	IF	Temp_Mirror.stat.lrTempK > cfg.lrTemp_Precooled	AND  
		Pressure_Cryo.stat.lrPressure >= cfg.lrPress_Atm  		THEN
		ctrl.bEnable_RepressCtrl	:= FALSE;
		// Disable Evacuation Valve control
		ctrl.bEnable_Evac	:= FALSE;
		M_SysLog('Re-pressurization complete. State is Warm-Pressurized.');
		stat.nState	:= E_CRYO_CTRL_STATE.WARM_PRESS;
	ELSIF NOT ctrl.bEnable_RepressCtrl THEN
		// Re-pressurization has been interrupted.
		// Go back to WARM_VACUUM state.
		M_SysLog('Re-pressurization interrupted. State is Warm-Vacuum.');
		stat.nState := E_CRYO_CTRL_STATE.WARM_VACUUM;
	END_IF
	M_SetStatus(stat.nState);	
	RETURN;
	
	
	/////////////////////////////////
	E_CRYO_CTRL_STATE.ERROR:
	/////////////////////////////////
	//
	// RESET the controller in order to try to clear error
	IF ctrl.bReset THEN
		ctrl.bReset	:= FALSE;	// Clear RESET flag
		// Goto NONE state
		stat.nState	:= E_CRYO_CTRL_STATE.NONE;
		M_SetStatus(stat.nState);	
	ELSIF NOT stat.bError  THEN
		// Goto NONE state
		stat.nState	:= E_CRYO_CTRL_STATE.NONE;
		M_SetStatus(stat.nState);	
	END_IF
	RETURN;

END_CASE
END_METHOD

METHOD M_SysLog
VAR_INPUT
	str:	STRING(80);
END_VAR
VAR
	i:	INT;
END_VAR
nLogPos	:= nLogPos + 1;
IF nLogPos > 9 THEN
	FOR i := 1 TO 9 DO
		// Shift last 9 readings
		ptrLog[i-1]^ := ptrLog[i]^;
	END_FOR
	nLogPos	:= 9;
END_IF

ptrLog[nLogPos]^ := str;
END_METHOD

END_FUNCTION_BLOCK

// ---- POUs/Actuators/FB_CRYO_LN2_CTRL.TcPOU
FUNCTION_BLOCK FB_CRYO_LN2_CTRL EXTENDS FB_CRYO_BIN_CTRL
VAR_INPUT
	in_lrTempK:		LREAL;			// Temperature input value [K]
	in_bValid:		BOOL := TRUE;	// Temperature Valid flag
	// Two parameters for decision making
	in_lrTempValveOpen:		LREAL := 91.27;		// Open  valve if temperature above this value [K]
	in_lrTempValveClose:	LREAL := 79.148;	// Close valve if temperature below this value [K]
END_VAR
VAR_OUTPUT
END_VAR
VAR
END_VAR

// Check the validity of the temperature reading.
// Start the check after 200 cycles.
IF stat.nCycleCounter > 200 THEN
	IF NOT in_bValid THEN
		// The temperature is not valid. 
		// The controller cannot work.
		stat.bCtrlOK	:= FALSE;
	ELSIF in_lrTempValveClose >= in_lrTempValveOpen THEN
		// Wrong configuration.
		// ValveClose MUST be lower than ValveOpen temperature
		stat.bCtrlOK	:= FALSE;
	ELSE
		// The temperature is valid. 
		stat.bCtrlOK	:= TRUE;
	END_IF
ELSE
	// The temperature is valid. 
	stat.bCtrlOK	:= TRUE;
END_IF

// Execute parent FB.
SUPER^();

METHOD M_SetStatus
VAR_INPUT
	nState:	E_CRYO_BIN_CTRL_STATE;
END_VAR
// Execute the status of the parent FB
SUPER^.M_SetStatus(nState);

// Set proper error description, if any.
IF Actuator.stat.bError THEN
	stat.sState	:= 'Valve failure';
ELSIF NOT stat.bCtrlOK THEN
	stat.sState	:= 'Temperature not valid';
END_IF
END_METHOD

METHOD M_User_SetAction : INT
VAR_INPUT
END_VAR
// TODO USER
// Overwrite Method FB_CRYO_BIN_CTRL::M_User_SetOutput()
//
// This method implements the logic for controlling the LN2 valve.
// 
// FB_CRYO_LN2_CTRL input parameters:
//
// in_lrTempK          - LN2 temperature
// in_bValid           - Flag if temperature reading is valid
// in_lrTempValveOpen  - Temperature upper limit [K]. Valve opens  when:  LN2 > in_lrTempValveOpen
// in_lrTempValveClose - Temperature lower limit [K]. Valve closes when:  LN2 < in_lrTempValveClose
//
// in_lrTempValveOpen > in_lrTempValveClose, e.g. 91.27K > 79.148K.
//
	
IF	stat.nState = E_CRYO_BIN_CTRL_STATE.ACTIVE_OFF  OR  
	stat.nState = E_CRYO_BIN_CTRL_STATE.ACTIVE_ON THEN
	// Check if input temperature value is valid.
	// If OK, check temperature against the limits	
	IF NOT stat.bCtrlOK THEN
		// Temperature reading is not valid.
		// Dectivate the actuator, i.e. close the valve
		M_User_SetAction	:= E_CRYO_BIN_CTRL_ACTION.OFF;
		stat.nState	:= E_CRYO_BIN_CTRL_STATE.ERROR;
	ELSIF in_lrTempK > in_lrTempValveOpen THEN
		// Activate the actuator, i.e. open the valve
		M_User_SetAction	:= E_CRYO_BIN_CTRL_ACTION.ON;
	ELSIF in_lrTempK < in_lrTempValveClose THEN
		// Dectivate the actuator, i.e. close the valve
		M_User_SetAction	:= E_CRYO_BIN_CTRL_ACTION.OFF;
	END_IF
	
ELSE
	// Don't do anything
	M_User_SetAction	:= E_CRYO_BIN_CTRL_ACTION.NONE;
END_IF
END_METHOD

END_FUNCTION_BLOCK

// ---- POUs/Actuators/FB_CRYO_BIN_CTRL.TcPOU
// Binary Controller
FUNCTION_BLOCK FB_CRYO_BIN_CTRL
VAR_INPUT
	in_nFeedback:		E_CRYO_BIN_ACT_FEEDBACK := E_CRYO_BIN_ACT_FEEDBACK.ON_ONLY;	// Feedbacks
	in_nTimeout:		UDINT := 10000;	// Timeout for switching on/off [ms]. Default 10000.
	in_bActiveLowCtrl:	BOOL := FALSE;	// Active Low for Control output
	in_bActiveLowStat:	BOOL := FALSE;	// Active Low for Status signals, i.e. feedback
	in_bEnable:			BOOL := FALSE;	// Controller active while in_bEnable is TRUE
END_VAR
VAR
	
	{attribute 'OPC.UA.DA' := '1'}
	Actuator:	FB_CRYO_BIN_ACT;	// Heater, valve, etc.
	
	stat:		T_CRYO_BIN_CTRL_STATUS;


	{attribute 'OPC.UA.DA' := '0'}
	bReset:		BOOL := FALSE;		// RESET Command


	{attribute 'OPC.UA.DA' := '0'}
	timer:		TON;		// Timer for commands
	
	
END_VAR

// Increment cycle counter
stat.nCycleCounter := stat.nCycleCounter + 1;

// Execute Actuator FB on every cycle
Actuator(
	in_nFeedback		:= in_nFeedback,
	in_nTimeout			:= in_nTimeout,
	in_bActiveLowCtrl	:= in_bActiveLowCtrl,
	in_bActiveLowStat	:= in_bActiveLowStat);


CASE stat.nState OF
	/////////////////////////////////
	E_CRYO_BIN_CTRL_STATE.NONE:
	/////////////////////////////////
	//
	// This is the state on power-up.
	// Determine the initial state based on the command amd actuator state.
	IF Actuator.stat.bError  OR NOT stat.bCtrlOK	THEN
		stat.nState	:= E_CRYO_BIN_CTRL_STATE.ERROR;
	ELSIF in_bEnable  AND  Actuator.stat.bON	THEN
		stat.nState	:= E_CRYO_BIN_CTRL_STATE.ACTIVE_ON;
	ELSIF in_bEnable  AND  Actuator.stat.bOFF	THEN
		stat.nState	:= E_CRYO_BIN_CTRL_STATE.ACTIVE_OFF;
	ELSIF NOT in_bEnable  THEN
		stat.nState	:= E_CRYO_BIN_CTRL_STATE.OFF;
	END_IF
	M_SetStatus(stat.nState);	
	RETURN;
	

	/////////////////////////////////
	E_CRYO_BIN_CTRL_STATE.OFF:
	/////////////////////////////////
	//
	IF	Actuator.stat.bError	OR NOT stat.bCtrlOK	THEN
		stat.nState	:= E_CRYO_BIN_CTRL_STATE.ERROR;
	ELSIF in_bEnable  THEN
		// Activate the control loop.
		// Goto Active_Off first.
		//
		// Start the timer
		timer(IN:=FALSE);
		timer(IN:=TRUE, PT:=UDINT_TO_TIME(in_nTimeout));
		// Set next state
		stat.nState	:= E_CRYO_BIN_CTRL_STATE.ACTIVE_OFF;
	END_IF
	M_SetStatus(stat.nState);	
	RETURN;
	
	
	/////////////////////////////////
	E_CRYO_BIN_CTRL_STATE.ACTIVE_OFF:
	/////////////////////////////////
	//
	IF	Actuator.stat.bError	OR NOT stat.bCtrlOK  THEN
		stat.nState	:= E_CRYO_BIN_CTRL_STATE.ERROR;
	ELSIF NOT in_bEnable  THEN
		// Goto Off.
		//
		// Set next state
		stat.nState	:= E_CRYO_BIN_CTRL_STATE.OFF;
	ELSIF M_User_SetAction() = E_CRYO_BIN_CTRL_ACTION.ON THEN
		// Goto Active_Off.
		//
		// Start the timer
		timer(IN:=FALSE);
		timer(IN:=TRUE, PT:=UDINT_TO_TIME(in_nTimeout));
		
		// Trigger action
		Actuator(in_bExecute:=FALSE);
		Actuator(in_bExecute:=TRUE, in_nCommand:=E_CRYO_BIN_ACT_CMD.ON);
		
		// Set next state
		stat.nState	:= E_CRYO_BIN_CTRL_STATE.ACTIVE_SWITCHING_ON;
	END_IF
	M_SetStatus(stat.nState);	
	RETURN;
	
	
	//////////////////////////////////////////
	E_CRYO_BIN_CTRL_STATE.ACTIVE_SWITCHING_ON:
	//////////////////////////////////////////
	//
	// Check for timeout
	timer(IN:=TRUE);
	IF timer.Q THEN
		// Stop the timer
		timer(IN:=FALSE);
		// Goto ERROR state
		stat.nState	:= E_CRYO_BIN_CTRL_STATE.ERROR;
	ELSIF	Actuator.stat.bError	THEN
		stat.nState	:= E_CRYO_BIN_CTRL_STATE.ERROR;
	ELSIF Actuator.stat.bON THEN
		// The actuator is ON, transition completed.
		// Goto Active_On.
		stat.nState	:= E_CRYO_BIN_CTRL_STATE.ACTIVE_ON;
	END_IF
	M_SetStatus(stat.nState);	
	RETURN;
	

	/////////////////////////////////
	E_CRYO_BIN_CTRL_STATE.ACTIVE_ON:
	/////////////////////////////////
	//
	IF	Actuator.stat.bError	THEN
		stat.nState	:= E_CRYO_BIN_CTRL_STATE.ERROR;
	ELSIF	NOT in_bEnable 		OR  
			NOT stat.bCtrlOK	OR
			M_User_SetAction() = E_CRYO_BIN_CTRL_ACTION.OFF THEN
		// Goto Active_Off.
		// If NOT in_bExecute, the system will continue to complete OFF
		//
		// Start the timer
		timer(IN:=FALSE);
		timer(IN:=TRUE, PT:=UDINT_TO_TIME(in_nTimeout));
		
		// Trigger action
		Actuator(in_bExecute:=FALSE);
		Actuator(in_bExecute:=TRUE, in_nCommand:=E_CRYO_BIN_ACT_CMD.OFF);
		
		// Set next state
		stat.nState	:= E_CRYO_BIN_CTRL_STATE.ACTIVE_SWITCHING_OFF;
	END_IF
	M_SetStatus(stat.nState);	
	RETURN;
	
	
	///////////////////////////////////////////
	E_CRYO_BIN_CTRL_STATE.ACTIVE_SWITCHING_OFF:
	///////////////////////////////////////////
	//
	// Check for timeout
	timer(IN:=TRUE);
	IF timer.Q THEN
		// Stop the timer
		timer(IN:=FALSE);
		// Goto ERROR state
		stat.nState	:= E_CRYO_BIN_CTRL_STATE.ERROR;
	ELSIF	Actuator.stat.bError	THEN
		stat.nState	:= E_CRYO_BIN_CTRL_STATE.ERROR;
	ELSIF Actuator.stat.bOFF THEN
		// The actuator is OFF, transition completed.
		// Goto Active_Off.
		stat.nState	:= E_CRYO_BIN_CTRL_STATE.ACTIVE_OFF;
	END_IF
	M_SetStatus(stat.nState);	
	RETURN;
	
	/////////////////////////////////
	E_CRYO_BIN_CTRL_STATE.ERROR:
	/////////////////////////////////
	//
	M_User_TryRecovery();

END_CASE

METHOD M_Reset
VAR_INPUT
END_VAR
// By setting the bReset flag,
// The actuator will try to exit error state.
// In ERROR state, method M_User_TryRecovery() is executed.
bReset	:= TRUE;
END_METHOD

METHOD M_SetStatus
VAR_INPUT
	nState:	E_CRYO_BIN_CTRL_STATE;
END_VAR
stat.bActON		:= Actuator.stat.bON;
stat.bActOFF	:= Actuator.stat.bOFF;


CASE nState OF
	
	E_CRYO_BIN_CTRL_STATE.OFF:
	stat.bDone	:= TRUE;
	stat.bBusy	:= FALSE;
	stat.bError	:= FALSE;
	stat.bActive:= FALSE;
	stat.sState	:= 'OFF';
	
	E_CRYO_BIN_CTRL_STATE.ACTIVE_OFF:
	stat.bDone	:= TRUE;
	stat.bBusy	:= FALSE;
	stat.bError	:= FALSE;
	stat.bActive:= TRUE;
	stat.sState	:= 'ACTIVE_OFF';
	
	E_CRYO_BIN_CTRL_STATE.ACTIVE_ON:
	stat.bDone	:= TRUE;
	stat.bBusy	:= FALSE;
	stat.bError	:= FALSE;
	stat.bActive:= TRUE;
	stat.sState	:= 'ACTIVE_ON';
	
	E_CRYO_BIN_CTRL_STATE.ACTIVE_SWITCHING_ON:
	stat.bDone	:= FALSE;
	stat.bBusy	:= TRUE;
	stat.bError	:= FALSE;
	stat.bActive:= TRUE;
	stat.sState	:= 'ACTIVE_SWITCHING_ON...';
	
	E_CRYO_BIN_CTRL_STATE.ACTIVE_SWITCHING_OFF:
	stat.bDone	:= FALSE;
	stat.bBusy	:= TRUE;
	stat.bError	:= FALSE;
	stat.bActive:= TRUE;
	stat.sState	:= 'ACTIVE_SWITCHING_OFF...';
	
	E_CRYO_BIN_CTRL_STATE.ERROR:
	stat.bDone	:= TRUE;
	stat.bBusy	:= FALSE;
	stat.bError	:= TRUE;
	stat.bActive:= FALSE;
	stat.sState	:= 'ERROR';

END_CASE
END_METHOD

METHOD M_User_SetAction : INT
VAR_INPUT
END_VAR
// TODO USER
//
// This method implements the logic for controlling the actuator.
// The actuator can be a heater, valve, etc.
// There are two input values from sensors and two deltas for comparison.
//
// This example implements the heater control with the following assumptions:
//
// in_lrInput1 - Temperature of the Cryo Bench (B)
// in_lrInput2 - Temperature of the Detector (D). Coming from Lakeshore.
// in_lrPar1 - Delta [K] to turn the heater ON:  IF B < D - in_lrPar1
// in_lrPar2 - Delta [K] to turn the heater OFF: IF B > D - in_lrPar2
//
// in_lrDelta1 > in_lrDelta2, e.g. 10K > 4K.
//
IF	stat.nState = E_CRYO_BIN_CTRL_STATE.ACTIVE_OFF  OR  
	stat.nState = E_CRYO_BIN_CTRL_STATE.ACTIVE_ON THEN
(*	
	IF in_lrInput1 < in_lrInput2 - in_lrPar1 THEN
		// Activate the actuator
		M_User_SetOutput	:= E_CRYO_BIN_CTRL_ACTION.ON;
	ELSIF in_lrInput1 > in_lrInput2 - in_lrPar2 THEN
		// Dectivate the actuator
		M_User_SetOutput	:= E_CRYO_BIN_CTRL_ACTION.OFF;
	END_IF
*)
ELSE
	// Don't do anything
	M_User_SetAction	:= E_CRYO_BIN_CTRL_ACTION.NONE;
END_IF
END_METHOD

METHOD M_User_TryRecovery
VAR_INPUT
END_VAR
// TODO USER
// This is the default recovery routine.
// To be customided by the user, if needed.
//
IF bReset THEN
	// RESET the controller in order to try to clear error
	bReset	:= FALSE;	// Clear RESET flag
	
	// Start the timer
	timer(IN:=FALSE);
	timer(IN:=TRUE, PT:=T#5S);
	
	// Trigger action
	Actuator(in_bExecute:=FALSE);
	Actuator(in_bExecute:=TRUE, in_nCommand:=E_CRYO_BIN_ACT_CMD.OFF);
	
	// Goto SWITCHING_OFF state
	stat.nState	:= E_CRYO_BIN_CTRL_STATE.ACTIVE_SWITCHING_OFF;
	M_SetStatus(stat.nState);	
ELSIF NOT Actuator.stat.bError AND stat.bCtrlOK  THEN
	// Self recovery since everything seems to be OK now.
	// Goto NONE state.
	// From there proper state will be found and set.
	stat.nState	:= E_CRYO_BIN_CTRL_STATE.NONE;
	M_SetStatus(stat.nState);	
END_IF
END_METHOD

END_FUNCTION_BLOCK

// ---- POUs/Actuators/FB_CRYO_BIN_ACT.TcPOU
FUNCTION_BLOCK FB_CRYO_BIN_ACT
VAR_INPUT
	in_nFeedback:		E_CRYO_BIN_ACT_FEEDBACK := E_CRYO_BIN_ACT_FEEDBACK.ON_ONLY;	// Feedback configuration.
	in_nTimeout:		UDINT := 10000;	// Timeout for switching on/off [ms]. Default 10000.
	in_bActiveLowCtrl:	BOOL := FALSE;	// Active Low for Control output
	in_bActiveLowStat:	BOOL := FALSE;	// Active Low for Status signals, i.e. feedback
	in_nCommand:		E_CRYO_BIN_ACT_CMD	:= E_CRYO_BIN_ACT_CMD.NONE;	// Command
	in_bExecute:		BOOL := FALSE;	// Execute trigger
END_VAR
VAR
	{attribute 'OPC.UA.DA' := '0'}
	i_nCouplerState	AT%I*:	UINT;		// Terminal state. Should be 8, i.e. OP.
	{attribute 'OPC.UA.DA' := '0'}
	i_bON			AT%I*:	BOOL;		// Feedback for ON
	{attribute 'OPC.UA.DA' := '0'}
	i_bOFF			AT%I*:	BOOL;		// Feedback for OFF
	
	{attribute 'OPC.UA.DA' := '0'}
	q_bCtrl			AT%Q*:	BOOL;		// Control output signal
	
	stat:		T_CRYO_BIN_ACT_STATUS;

	
	{attribute 'OPC.UA.DA' := '0'}
	timer:		TON;		// Timer for commands
	{attribute 'OPC.UA.DA' := '0'}
	trigCMD:	R_TRIG;		// Trigger for new command
	
	{attribute 'OPC.UA.DA' := '0'}
	nCommand:	E_CRYO_BIN_ACT_CMD	:= E_CRYO_BIN_ACT_CMD.NONE;	// Command

END_VAR

// Get the feedback
M_GetFeedback();

// Check for new command
trigCMD(CLK:=in_bExecute);
IF trigCMD.Q THEN
	nCommand			:= in_nCommand;
	stat.nLastCommand	:= in_nCommand;
ELSE
	nCommand		:= E_CRYO_BIN_ACT_CMD.NONE;
END_IF

// If the system is not operational, this is an error.
IF i_nCouplerState <> 8 THEN
	stat.nState	:= E_CRYO_BIN_ACT_STATE.ERROR;
	stat.sState	:= 'ERROR: System not OPERATIONAL';
	M_SetStatus(stat.nState);	
END_IF

CASE stat.nState OF
	/////////////////////////////////
	E_CRYO_BIN_ACT_STATE.NONE:
	/////////////////////////////////
	//
	// Determine the initial state based on the feedback
	IF stat.bON	THEN
		stat.nState	:= E_CRYO_BIN_ACT_STATE.ON;
	ELSIF stat.bOFF	THEN
		stat.nState	:= E_CRYO_BIN_ACT_STATE.OFF;
	ELSE
		stat.nState	:= E_CRYO_BIN_ACT_STATE.ERROR;
		stat.sState	:= 'ERROR';
	END_IF
	M_SetStatus(stat.nState);	
	RETURN;
	

	/////////////////////////////////
	E_CRYO_BIN_ACT_STATE.OFF:
	/////////////////////////////////
	//
	IF	stat.bON  OR  
		stat.bError	THEN
		// This should never happen in state OFF
		stat.nState	:= E_CRYO_BIN_ACT_STATE.ERROR;
		stat.sState	:= 'ERROR: Lost ON state.';
		M_SetStatus(stat.nState);	
	ELSE
		// Check for command to go ON
		IF nCommand = E_CRYO_BIN_ACT_CMD.ON THEN
			// Start the timer
			timer(IN:=FALSE);
			timer(IN:=TRUE, PT:=UDINT_TO_TIME(in_nTimeout));
			// Activate the output
			M_SetCtrlOutput(TRUE);
			// Goto SWITCHING_ON state
			stat.nState	:= E_CRYO_BIN_ACT_STATE.SWITCHING_ON;
			M_SetStatus(stat.nState);	
		END_IF
	END_IF
	RETURN;
	
	
	/////////////////////////////////
	E_CRYO_BIN_ACT_STATE.SWITCHING_ON:
	/////////////////////////////////
	//
	// Check for timeout
	timer(IN:=TRUE);
	IF timer.Q THEN
		// Stop the timer
		timer(IN:=FALSE);
		// Goto ERROR state
		stat.nState	:= E_CRYO_BIN_ACT_STATE.ERROR;
		stat.sState	:= 'ERROR: Timeout switching ON';
		M_SetStatus(stat.nState);	
		RETURN;
	END_IF
	
	// Check if we have reached ON state
	IF stat.bON	AND NOT stat.bOFF	THEN
		// Stop the timer
		timer(IN:=FALSE);
		// Goto ON state
		stat.nState	:= E_CRYO_BIN_ACT_STATE.ON;
		M_SetStatus(stat.nState);	
	END_IF
	RETURN;
	

	/////////////////////////////////
	E_CRYO_BIN_ACT_STATE.ON:
	/////////////////////////////////
	//
	IF	stat.bOFF  OR  
		stat.bError	THEN
		// This should never happen in state ON
		stat.nState	:= E_CRYO_BIN_ACT_STATE.ERROR;
		stat.sState	:= 'ERROR: Lost OFF state.';
		M_SetStatus(stat.nState);	
	ELSE
		// Check for command to go OFF
		IF nCommand = E_CRYO_BIN_ACT_CMD.OFF THEN
			// Start the timer
			timer(IN:=FALSE);
			timer(IN:=TRUE, PT:=UDINT_TO_TIME(in_nTimeout));
			// Deactivate the output
			M_SetCtrlOutput(FALSE);
			// Goto SWITCHING_OFF state
			stat.nState	:= E_CRYO_BIN_ACT_STATE.SWITCHING_OFF;
			M_SetStatus(stat.nState);	
		END_IF
	END_IF
	RETURN;
	
	
	//////////////////////////////////
	E_CRYO_BIN_ACT_STATE.SWITCHING_OFF:
	//////////////////////////////////
	//
	// Check for timeout
	timer(IN:=TRUE);
	IF timer.Q THEN
		// Stop the timer
		timer(IN:=FALSE);
		// Goto ERROR state
		stat.nState	:= E_CRYO_BIN_ACT_STATE.ERROR;
		stat.sState	:= 'ERROR: Timeout switching OFF';
		M_SetStatus(stat.nState);	
		RETURN;
	END_IF
	
	// Check if we have reached OFF state
	IF stat.bOFF AND NOT stat.bON	THEN
		// Stop the timer
		timer(IN:=FALSE);
		// Goto OFF state
		stat.nState	:= E_CRYO_BIN_ACT_STATE.OFF;
		M_SetStatus(stat.nState);	
	END_IF
	RETURN;
	
	/////////////////////////////////
	E_CRYO_BIN_ACT_STATE.ERROR:
	/////////////////////////////////
	//
	// Deactivate the output
	M_SetCtrlOutput(FALSE);
	
	// Check for command to go ON
	IF nCommand = E_CRYO_BIN_ACT_CMD.ON THEN
		// Start the timer
		timer(IN:=FALSE);
		timer(IN:=TRUE, PT:=UDINT_TO_TIME(in_nTimeout));
		// Activate the output
		M_SetCtrlOutput(TRUE);
		// Goto SWITCHING_ON state
		stat.nState	:= E_CRYO_BIN_ACT_STATE.SWITCHING_ON;
		M_SetStatus(stat.nState);	
	// Check for command to go OFF
	ELSIF nCommand = E_CRYO_BIN_ACT_CMD.OFF THEN
		// Start the timer
		timer(IN:=FALSE);
		timer(IN:=TRUE, PT:=UDINT_TO_TIME(in_nTimeout));
		// Deactivate the output
		M_SetCtrlOutput(FALSE);
		// Goto SWITCHING_OFF state
		stat.nState	:= E_CRYO_BIN_ACT_STATE.SWITCHING_OFF;
		M_SetStatus(stat.nState);	
	END_IF
	RETURN;

END_CASE

METHOD M_GetFeedback
VAR_INPUT
END_VAR
// Get ON/OFF status based on active low configuration
IF in_bActiveLowStat	THEN
	stat.bON	:= NOT i_bON;
	stat.bOFF	:= NOT i_bOFF;
ELSE
	stat.bON	:= i_bON;
	stat.bOFF	:= i_bOFF;
END_IF

// Check for possible feedback errors.
// Also, adjust the OFF signal, if only ON feedback exists.
IF in_nFeedback = E_CRYO_BIN_ACT_FEEDBACK.ON_AND_OFF  THEN
	// There are separate signals for ON and OFF.
	// The status is already properly assigned. Nothing more to do.
	// If both feedback signals are active, this is an error.
	(*
	IF stat.bON AND stat.bOFF	THEN
		stat.nState	:= E_CRYO_BIN_ACT_STATE.ERROR;
		stat.sState	:= 'ERROR: Both ON and OFF signals active!';
		M_SetStatus(stat.nState);	
	END_IF
	*)
	;
ELSIF in_nFeedback = E_CRYO_BIN_ACT_FEEDBACK.ON_ONLY  THEN
	// There is only a feedback signal for ON.
	// Therefore, stat.bOFF := NOT stat.bON
	stat.bOFF	:= NOT stat.bON;
END_IF
END_METHOD

METHOD M_SetCtrlOutput
VAR_INPUT
	in_bSignal:	BOOL;
END_VAR
// Set control output signal based on active low configuration
IF in_bActiveLowCtrl	THEN
	q_bCtrl	:= NOT in_bSignal;
ELSE
	q_bCtrl	:= in_bSignal;
END_IF
END_METHOD

METHOD M_SetStatus
VAR_INPUT
	nState:	E_CRYO_BIN_ACT_STATE;
END_VAR
CASE stat.nState OF
	
	E_CRYO_BIN_ACT_STATE.OFF,
	E_CRYO_BIN_ACT_STATE.ON:
	stat.bDone	:= TRUE;
	stat.bBusy	:= FALSE;
	stat.bError	:= FALSE;
	
	E_CRYO_BIN_ACT_STATE.SWITCHING_ON,
	E_CRYO_BIN_ACT_STATE.SWITCHING_OFF:
	stat.bDone	:= FALSE;
	stat.bBusy	:= TRUE;
	stat.bError	:= FALSE;
	
	E_CRYO_BIN_ACT_STATE.ERROR:
	stat.bDone	:= TRUE;
	stat.bBusy	:= FALSE;
	stat.bError	:= TRUE;
END_CASE

// Set status string
CASE stat.nState OF
	
	E_CRYO_BIN_ACT_STATE.OFF:
	stat.sState	:= 'OFF';
	
	E_CRYO_BIN_ACT_STATE.ON:
	stat.sState	:= 'ON';
	
	E_CRYO_BIN_ACT_STATE.SWITCHING_ON:
	stat.sState	:= 'SWITCHING_ON...';
	
	E_CRYO_BIN_ACT_STATE.SWITCHING_OFF:
	stat.sState	:= 'SWITCHING_OFF...';
	
	E_CRYO_BIN_ACT_STATE.ERROR:
	// Error string was set where the error was detected.
	//	stat.sState	:= 'ERROR';
	;
END_CASE
END_METHOD

END_FUNCTION_BLOCK

// ---- POUs/Actuators/FB_CRYO_VALVE_CTRL.TcPOU
FUNCTION_BLOCK FB_CRYO_VALVE_CTRL EXTENDS FB_CRYO_BIN_CTRL
VAR_INPUT
END_VAR
VAR_OUTPUT
END_VAR
VAR
END_VAR

// Execute parent FB.
SUPER^();

METHOD M_SetStatus
VAR_INPUT
	nState:	E_CRYO_BIN_CTRL_STATE;
END_VAR
// Execute the status of the parent FB
SUPER^.M_SetStatus(nState);

// Set proper error description, if any.
IF Actuator.stat.bError THEN
	stat.sState	:= 'Valve failure';
END_IF
END_METHOD

METHOD M_User_SetAction : INT
VAR_INPUT
END_VAR
// TODO USER
// Set Valve command based on the input parameter in_bEnable.
//
	
IF	stat.nState = E_CRYO_BIN_CTRL_STATE.ACTIVE_OFF  AND in_bEnable THEN
	// Activate the actuator, i.e. open the valve
	M_User_SetAction	:= E_CRYO_BIN_CTRL_ACTION.ON;
ELSIF  stat.nState = E_CRYO_BIN_CTRL_STATE.ACTIVE_ON AND NOT in_bEnable THEN
	// Dectivate the actuator, i.e. close the valve
	M_User_SetAction	:= E_CRYO_BIN_CTRL_ACTION.OFF;
ELSE
	// Don't do anything
	M_User_SetAction	:= E_CRYO_BIN_CTRL_ACTION.NONE;
END_IF
END_METHOD

END_FUNCTION_BLOCK

// ---- POUs/Subsystems/Evacuation/FB_CRYO_EVACUATION_SYSTEM.TcPOU
//
// Evacuation System Controller.
// The system consists of:
// - Evacuation Valve
// - Root Pump
// - Turbo Pump
//
FUNCTION_BLOCK FB_CRYO_EVACUATION_SYSTEM
VAR_INPUT
	in_Cryo_Cfg:			T_CRYO_CFG;					// Cryo configuration
	in_Temp_Cryo:			T_CRYO_TEMPERATURE_STATUS;	// Cold Bench temperature	
	in_Pressure_Cryo:		T_CRYO_PRESSURE_STATUS;		// Cryostat Pressure
	in_Pressure_Evac:		T_CRYO_PRESSURE_STATUS;		// Evacuation Pressure
	
	in_bRepressValveOpen:	BOOL;	// Repressure Valve Open flag
	in_bRepressValveOK:		BOOL;	// Repressure Valve OK flag
	in_nFeedback:	E_CRYO_BIN_ACT_FEEDBACK := E_CRYO_BIN_ACT_FEEDBACK.ON_ONLY;	// Feedbacks
	// Time between closing Vac valve and Switching OFF the vac Pump [ms]
	in_nTimeout:	UDINT := 3200;	// Timeout for switching on/off [ms]
	in_bEnable:		BOOL := FALSE;	// Controller active while in_bEnable is TRUE
	in_bCmd:		BOOL := FALSE;	// ON=TRUE, OFF=FALSE
END_VAR
VAR
	
	{attribute 'OPC.UA.DA' := '0'}
	i_bRootPumpOn	AT%I*:	BOOL;		// Root Pump Feedback
	{attribute 'OPC.UA.DA' := '0'}
	i_bTurboPumpOn	AT%I*:	BOOL;		// Turbo Pump Feedback
	
	{attribute 'OPC.UA.DA' := '0'}
	q_bPumpCtrl		AT%Q*:	BOOL;			// Pump Control signal
	
	stat:			T_CRYO_EVACUATION_SYSTEM_STATUS;

	{attribute 'OPC.UA.DA' := '1'}
	Valve:	FB_CRYO_BIN_ACT;			// Evacuation Valve 

	{attribute 'OPC.UA.DA' := '0'}
	bExecute_Valve:	BOOL := FALSE;

	{attribute 'OPC.UA.DA' := '0'}
	nCommand_Valve:	E_CRYO_BIN_ACT_CMD	:= E_CRYO_BIN_ACT_CMD.NONE;	// Command

	{attribute 'OPC.UA.DA' := '0'}
	bReset:		BOOL := FALSE;		// RESET Command

	{attribute 'OPC.UA.DA' := '0'}
	bValveCmd:	BOOL := FALSE;		// Valve Command - TRUE=OPEN, FALSE=CLOSE


	{attribute 'OPC.UA.DA' := '0'}
	timerTurbo:	TON;		// Timer for Turbo Pump
	
	{attribute 'OPC.UA.DA' := '0'}
	timerValveDelay:	TON;		// Timer for measuring time after Valve is closed
	
	{attribute 'OPC.UA.DA' := '0'}
	timerValveCtrl:	TON;		// Timer for Valve open/close timeout
	
	{attribute 'OPC.UA.DA' := '0'}
	trigEnable:	R_TRIG;			// Trigger for in_bEnable
	
	{attribute 'OPC.UA.DA' := '0'}
	trigDisable:F_TRIG;			// Trigger for in_bEnable=FALSE, i.e. Disable
	
	{attribute 'OPC.UA.DA' := '0'}
	trigTurbo:	R_TRIG;		// Trigger for start of TurboPump
	
	{attribute 'OPC.UA.DA' := '0'}
	trigValveClosed:	R_TRIG;		// Trigger for Valve Closed. Start timerValve on trigger.
	
END_VAR

// Increment cycle counter
stat.nCycleCounter := stat.nCycleCounter + 1;

// Pump control based on Valve status.
M_PumpCtrl();

// Check for errors
M_CheckErrors();

// Get Valve Command based on pressure and temperature conditions
M_SetValveCommand();


// Execute Valve FB on every cycle
Valve(	in_bExecute	:= bExecute_Valve,
		in_nCommand	:= nCommand_Valve,
		in_nFeedback:= in_nFeedback);


M_StateMachine();

METHOD M_CheckErrors
VAR_INPUT
END_VAR
VAR
END_VAR
// TODO: Set stat.sStatus for each failure
IF Valve.stat.bON  AND  (in_bRepressValveOpen  OR  NOT in_bRepressValveOK) THEN
	// Emergency situation. Close the Valve
	stat.bEmergency	:= TRUE;
	stat.bError	:= TRUE;
ELSIF stat.bEnabled  AND  (in_bRepressValveOpen  OR  NOT in_bRepressValveOK) THEN
	// The Evacuation system should never be enabled 
	// if there is a problem with the repressurizing valve.
	// Emergency situation. Do not operate.
	stat.bEmergency	:= TRUE;
	stat.bError	:= TRUE;
ELSIF NOT in_bRepressValveOK THEN
	stat.bError	:= TRUE;
ELSIF NOT in_Pressure_Cryo.bValid THEN
	stat.bError	:= TRUE;
ELSIF NOT in_Pressure_Evac.bValid THEN
	stat.bError	:= TRUE;
ELSIF Valve.stat.bError THEN
	stat.bError	:= TRUE;
ELSE
	stat.bError	:= FALSE;
END_IF

// Additional check for emergency situation.
// If there is an error while the Evacuation Valve is open, close it immediately.
IF stat.bError  AND  Valve.stat.bON  THEN
	stat.bEmergency	:= TRUE;
END_IF

IF stat.bError  THEN
	stat.bEnabled	:= FALSE;	// Disable Evacuation System
END_IF
END_METHOD

// Pump control based on Valve status.
METHOD M_PumpCtrl
VAR_INPUT
END_VAR
//
// Capture in_bEnable going TRUE.
// When it happens, start the pumps by activating the control output.
//
trigEnable(CLK:=in_bEnable);
IF trigEnable.Q THEN
	stat.bEnabled	:= TRUE;
	stat.bEmergency	:= FALSE;	// Clear emergency warning, if any
	stat.bError		:= FALSE;	// Clear error
	q_bPumpCtrl		:= TRUE;	// Start pumps
ELSIF NOT in_bEnable THEN
	stat.bEnabled		:= FALSE;
END_IF


//
// Set the status of the Root Pump
//
stat.bRootPumpON	:= i_bRootPumpOn;


//
// Set the status of the Turbo Pump
//
IF i_bTurboPumpOn THEN
	// Turbo pump is running.
	stat.bTurboPumpON	:= TRUE;
ELSE
	timerTurbo(IN:=FALSE);
	stat.bTurboPumpON		:= FALSE;
	stat.bTurboPump10min	:= FALSE;
END_IF



//
// Capture the moment when Turbo Pump started.
// Turbo Pump is fully operational after 10 min of operation (in_nTime_TurboPump).
//
// Execute timer for Turbo Pump
timerTurbo();

trigTurbo(CLK:=stat.bTurboPumpON);
IF trigTurbo.Q  THEN
	//
	// Turbo Pump has just started.
	// Start the timer that will signal that the turbo pump is fully operational.
	//
	// Reset the timer.
	timerTurbo(IN:=FALSE);
	// Start the timer for Turbo Pump warmup.
	timerTurbo(IN:=TRUE,PT:=UDINT_TO_TIME(in_Cryo_Cfg.nTime_TurboPump));
END_IF

IF timerTurbo.Q THEN
	// Turbo Pump is now fully operational.
	stat.bTurboPump10min	:= TRUE;
END_IF


//
// Capture the moment when the Valve is closed or the system is disabled.
// Pumps should be stopped in_nTime_DeltaTValve [ms] (e.g. 2000ms) after this event.
//
// Execute timer for Valve timer
timerValveDelay();


//
// Capture the moment when the valve is closed.
// Start the delay timer for in_Cryo_Cfg.nTime_DeltaTValve ms.
// After the delay, it is safe to stop the pumps.
//
trigValveClosed(CLK:=NOT stat.bValveOpen);
trigDisable(CLK:=stat.bEnabled);	// Falling edge of bEnable
IF trigValveClosed.Q OR trigDisable.Q  THEN
	// Reset the timer
	timerValveDelay(IN:=FALSE);
	// Start the Valve timer.
	timerValveDelay(IN:=TRUE,PT:=UDINT_TO_TIME(in_Cryo_Cfg.nTime_DeltaTValve));
END_IF


//
// The delay timer has expired.
// It is safe to stop the pumps.
//
IF timerValveDelay.Q THEN
	// Reset the timer
	timerValveDelay(IN:=FALSE);
	// Stop the pumps if evacuation is disabled
	IF NOT stat.bEnabled THEN
		q_bPumpCtrl	:= FALSE;
	END_IF
END_IF

// Update output var
stat.bValveOpen	:= Valve.stat.bON;
END_METHOD

METHOD M_SetStatus
VAR_INPUT
	nState:	E_CRYO_EVAC_SYS_STATE;
END_VAR
// TODO: Complete this


CASE nState OF
	
	E_CRYO_EVAC_SYS_STATE.OFF:
	stat.bDone	:= TRUE;
	stat.bBusy	:= FALSE;
	IF NOT stat.bError THEN
		stat.sState	:= 'OFF';
	END_IF
	stat.bActive	:= FALSE;
	
	E_CRYO_EVAC_SYS_STATE.ACTIVE_CLOSED:
	stat.bDone	:= TRUE;
	stat.bBusy	:= FALSE;
	IF NOT stat.bError THEN
		stat.sState	:= 'ACTIVE_OFF';
	END_IF
	stat.bActive	:= TRUE;
	
	E_CRYO_EVAC_SYS_STATE.ACTIVE_OPEN:
	stat.bDone	:= TRUE;
	stat.bBusy	:= FALSE;
	stat.bError	:= FALSE;
	stat.bActive	:= TRUE;
	stat.sState	:= 'ACTIVE_ON';
	
	E_CRYO_EVAC_SYS_STATE.ACTIVE_OPENING:
	stat.bDone	:= FALSE;
	stat.bBusy	:= TRUE;
	stat.bError	:= FALSE;
	stat.bActive	:= TRUE;
	stat.sState	:= 'ACTIVE_SWITCHING_ON...';
	
	E_CRYO_EVAC_SYS_STATE.ACTIVE_CLOSING:
	stat.bDone	:= FALSE;
	stat.bBusy	:= TRUE;
	stat.bError	:= FALSE;
	stat.bActive	:= TRUE;
	stat.sState	:= 'ACTIVE_SWITCHING_OFF...';
	
	E_CRYO_EVAC_SYS_STATE.ERROR:
	stat.bDone	:= TRUE;
	stat.bBusy	:= FALSE;
//	stat.bError	:= TRUE;
	stat.bActive	:= FALSE;
//	stat.sState	:= 'ERROR';

END_CASE
END_METHOD

//
// Determines if the valve should be open or closed.
// It sets the internal variable nCommand_Valve.
//
METHOD M_SetValveCommand
VAR_INPUT
END_VAR
// Reset bExecute_Valve flag and the Valve command.
// They might be set again depending on the bEnable flag and the environmental conditions.
bExecute_Valve	:= FALSE;
nCommand_Valve	:= E_CRYO_BIN_ACT_CMD.NONE;


// 
// Set the Valve command based on temperature and pressure.
// If the system is not enabled or there is an error, the valve should be closed.
//
IF stat.bError THEN
	// Close the Valve on any error.
	nCommand_Valve	:= E_CRYO_BIN_ACT_CMD.OFF;
ELSIF NOT stat.bEnabled THEN
	// Close the Valve if the system is Disabled/OFF.
	nCommand_Valve	:= E_CRYO_BIN_ACT_CMD.OFF;
ELSIF 	(in_Pressure_Cryo.lrPressure > in_Cryo_Cfg.lrPress_Atm)  AND  
		(in_Temp_Cryo.lrTempK > in_Cryo_Cfg.lrTemp_Warm) THEN
	// Cryo is Warm and Pressurized - safe to open Valve.
	nCommand_Valve	:= E_CRYO_BIN_ACT_CMD.ON;
//ELSIF NOT in_Pressure_Cryo.bInVacuum THEN
ELSIF in_Pressure_Cryo.lrPressure >= in_Cryo_Cfg.lrPress_InVac THEN
	// If not in vacuum, it means the cryostat must be WARM.
	IF (in_Pressure_Evac.lrPressure < in_Pressure_Cryo.lrPressure) THEN
		nCommand_Valve	:= E_CRYO_BIN_ACT_CMD.ON;
	END_IF
ELSIF in_Temp_Cryo.lrTempK < in_Cryo_Cfg.lrTemp_Precooled THEN
	// Cryostat is COLD.
	IF ((in_Pressure_Evac.lrPressure < in_Pressure_Cryo.lrPressure) AND stat.bTurboPumpON) OR  
		(stat.bTurboPump10min AND in_Pressure_Evac.lrPressure < 7.0E-5) THEN
		nCommand_Valve	:= E_CRYO_BIN_ACT_CMD.ON;
	END_IF
//ELSIF in_Pressure_Cryo.bInVacuum THEN
ELSIF in_Pressure_Cryo.lrPressure < in_Cryo_Cfg.lrPress_InVac THEN
	// Cryostat is in vacuum.
	IF (in_Pressure_Evac.lrPressure < in_Pressure_Cryo.lrPressure)  AND stat.bTurboPumpON THEN
		nCommand_Valve	:= E_CRYO_BIN_ACT_CMD.ON;
	END_IF
END_IF


//
// Apply Valve command depending on the Evacuation System state.
// Update the State as well.
//
IF (stat.bError OR stat.bEmergency) AND stat.nState	<> E_CRYO_EVAC_SYS_STATE.ACTIVE_CLOSING THEN
	//
	// There is an error or emergency in the system. 
	// Close the valve. 
	//
	// Trigger Valve closing
	bExecute_Valve	:= TRUE;
	nCommand_Valve	:= E_CRYO_BIN_ACT_CMD.OFF;
	Valve(in_bExecute	:= FALSE);
	Valve(in_bExecute	:= TRUE, in_nCommand := nCommand_Valve);
	stat.nState	:= E_CRYO_EVAC_SYS_STATE.ACTIVE_CLOSING;
ELSIF stat.nState = E_CRYO_EVAC_SYS_STATE.ACTIVE_CLOSED  THEN 
	IF  nCommand_Valve = E_CRYO_BIN_ACT_CMD.ON THEN
		bExecute_Valve	:= TRUE;
		timerValveCtrl(IN:=FALSE);
		timerValveCtrl(IN:=TRUE, PT:=UDINT_TO_TIME(in_nTimeout));
		stat.nState	:= E_CRYO_EVAC_SYS_STATE.ACTIVE_OPENING;
	ELSE
		bExecute_Valve	:= FALSE;
		IF stat.bEnabled THEN
			stat.nState	:= E_CRYO_EVAC_SYS_STATE.ACTIVE_CLOSED;
		ELSE
			stat.nState	:= E_CRYO_EVAC_SYS_STATE.OFF;
		END_IF
	END_IF
ELSIF stat.nState	= E_CRYO_EVAC_SYS_STATE.ACTIVE_OPEN  THEN 
	IF  nCommand_Valve = E_CRYO_BIN_ACT_CMD.OFF  OR  NOT stat.bEnabled  THEN
		bExecute_Valve	:= TRUE;
		timerValveCtrl(IN:=FALSE);
		timerValveCtrl(IN:=TRUE, PT:=UDINT_TO_TIME(in_nTimeout));
		stat.nState	:= E_CRYO_EVAC_SYS_STATE.ACTIVE_CLOSING;
	ELSE
		bExecute_Valve	:= FALSE;
		stat.nState	:= E_CRYO_EVAC_SYS_STATE.ACTIVE_OPEN;
	END_IF
END_IF
END_METHOD

METHOD M_StateMachine
VAR_INPUT
END_VAR
CASE stat.nState OF
	/////////////////////////////////
	E_CRYO_EVAC_SYS_STATE.NONE:
	/////////////////////////////////
	//
	// This is the state on power-up.
	// Determine the initial state based on the command and actuator state.
	IF NOT stat.bEnabled THEN
		IF Valve.stat.bOFF  AND  NOT stat.bRootPumpON AND NOT stat.bTurboPumpON THEN
			stat.nState	:= E_CRYO_EVAC_SYS_STATE.OFF;
		END_IF
	ELSE
		IF	stat.bError	THEN
			IF Valve.stat.bON THEN
				stat.nState	:= E_CRYO_EVAC_SYS_STATE.EMERGENCY;
			ELSE
				stat.nState	:= E_CRYO_EVAC_SYS_STATE.ERROR;
			END_IF
			stat.nState	:= E_CRYO_EVAC_SYS_STATE.ERROR;
		ELSIF Valve.stat.bON THEN
			stat.nState	:= E_CRYO_EVAC_SYS_STATE.ACTIVE_OPEN;
		ELSIF Valve.stat.bOFF  THEN
			stat.nState	:= E_CRYO_EVAC_SYS_STATE.ACTIVE_CLOSED;
		END_IF
	END_IF
	M_SetStatus(stat.nState);	
	RETURN;
	

	/////////////////////////////////
	E_CRYO_EVAC_SYS_STATE.OFF:
	/////////////////////////////////
	//
	IF stat.bEnabled  THEN
		// Set next state.
		stat.nState	:= E_CRYO_EVAC_SYS_STATE.ACTIVE_CLOSED;
	END_IF
	M_SetStatus(stat.nState);	
	RETURN;
	
	
	////////////////////////////////////////
	E_CRYO_EVAC_SYS_STATE.ACTIVE_CLOSING:
	////////////////////////////////////////
	//
	timerValveCtrl();
	IF timerValveCtrl.Q THEN
		// Closing failure
		stat.bCtrlOK	:= FALSE;
		stat.sStatus	:= 'Valve failed to close';
		stat.bError	:= TRUE;
		stat.nState	:= E_CRYO_EVAC_SYS_STATE.ERROR;
	ELSIF NOT stat.bValveOpen THEN
		timerValveCtrl(IN:=FALSE);
		// Set next state.
		stat.nState	:= E_CRYO_EVAC_SYS_STATE.ACTIVE_CLOSED;
	END_IF
	M_SetStatus(stat.nState);	
	RETURN;
	
	
	////////////////////////////////////////
	E_CRYO_EVAC_SYS_STATE.ACTIVE_CLOSED:
	////////////////////////////////////////
	//
	IF	NOT stat.bEnabled  THEN
		// Set next state
		stat.nState	:= E_CRYO_EVAC_SYS_STATE.OFF;
	ELSIF stat.bValveOpen THEN
		// Set next state.
		stat.nState	:= E_CRYO_EVAC_SYS_STATE.ACTIVE_OPEN;
	END_IF
	M_SetStatus(stat.nState);	
	RETURN;
	
	
	////////////////////////////////////////
	E_CRYO_EVAC_SYS_STATE.ACTIVE_OPENING:
	////////////////////////////////////////
	//
	timerValveCtrl();
	IF timerValveCtrl.Q THEN
		// Closing failure
		stat.bCtrlOK	:= FALSE;
		stat.sStatus	:= 'Valve failed to open';
		stat.bError	:= TRUE;
		stat.nState	:= E_CRYO_EVAC_SYS_STATE.ERROR;
	ELSIF stat.bValveOpen THEN
		timerValveCtrl(IN:=FALSE);
		// Set next state.
		stat.nState	:= E_CRYO_EVAC_SYS_STATE.ACTIVE_OPEN;
	END_IF
	M_SetStatus(stat.nState);	
	RETURN;
	
	
	//////////////////////////////////////////
	E_CRYO_EVAC_SYS_STATE.ACTIVE_OPEN:
	//////////////////////////////////////////
	//
	IF NOT stat.bValveOpen THEN
		// Set next state.
		stat.nState	:= E_CRYO_EVAC_SYS_STATE.ACTIVE_CLOSED;
	END_IF
	M_SetStatus(stat.nState);	
	RETURN;
	

	///////////////////////////////////////////
	E_CRYO_EVAC_SYS_STATE.EMERGENCY:
	///////////////////////////////////////////
	//
	IF Valve.stat.bOFF THEN
		// The actuator is OFF, transition completed.
		// Goto Active_Off.
		stat.nState	:= E_CRYO_EVAC_SYS_STATE.ACTIVE_CLOSED;
	END_IF
	M_SetStatus(stat.nState);	
	RETURN;
	
	/////////////////////////////////
	E_CRYO_EVAC_SYS_STATE.ERROR:
	/////////////////////////////////
	//
	M_User_TryRecovery();

END_CASE
END_METHOD

METHOD M_TrgValveClosure : BOOL
VAR_INPUT
END_VAR
END_METHOD

METHOD M_User_TryRecovery
VAR_INPUT
END_VAR
// TODO USER
// This is the default recovery routine.
// To be customided by the user, if needed.
//
IF bReset THEN
	// RESET the controller in order to try to clear error
	bReset	:= FALSE;	// Clear RESET flag
	
	// Trigger action
	Valve(in_bExecute:=FALSE);
	Valve(in_bExecute:=TRUE, in_nCommand:=E_CRYO_BIN_ACT_CMD.OFF);
	
	// Goto SWITCHING_OFF state
	stat.nState	:= E_CRYO_EVAC_SYS_STATE.ACTIVE_CLOSING;
	M_SetStatus(stat.nState);	
ELSIF NOT Valve.stat.bError AND stat.bCtrlOK  THEN
	// Self recovery since everything seems to be OK now.
	// Goto NONE state.
	// From there proper state will be found and set.
	stat.nState	:= E_CRYO_EVAC_SYS_STATE.NONE;
	M_SetStatus(stat.nState);	
END_IF
END_METHOD

END_FUNCTION_BLOCK

// ---- POUs/Actuators/FB_CRYO_HEATER_CTRL.TcPOU
FUNCTION_BLOCK FB_CRYO_HEATER_CTRL EXTENDS FB_CRYO_BIN_CTRL
VAR_INPUT
	// Two input values for comparison
	in_lrTemp1:		LREAL;	// Lowest temperature in  cryostat
	in_lrTemp2:		LREAL;	// Detector temperature.
	// Input values Valid flag
	in_bValidTemp1:	BOOL;
	in_bValidTemp2:	BOOL;
	// Two parameters for decision making
	// Delat-T SetPoint between Detector and Coldbench during WarmUp
	in_lrDelta_Low:		LREAL	:= 10.0;
	// Delat-T SetPoint between Detector and Coldbench during WarmUp	
	in_lrDelta_High:	LREAL	:= 5.0;

END_VAR
VAR_OUTPUT
END_VAR
VAR
END_VAR

// Set generic error if temperature inputs are not valid
IF NOT in_bValidTemp1 OR NOT in_bValidTemp2  THEN
	stat.bCtrlOK	:= FALSE;
ELSE
	stat.bCtrlOK	:= TRUE;
END_IF

// Execute parent FB.
SUPER^();

METHOD M_User_SetAction : INT
VAR_INPUT
END_VAR
// TODO USER
//
// This method implements the logic for controlling a heater.
// There are two input values from sensors and two deltas for comparison.
//
// This example implements the heater control with the following assumptions:
//
// in_lrTemp1 - Lowest Temperature in the system (L)
// in_lrTemp2 - Temperature of the Detector (D). Coming from Lakeshore.
//
// The heater should keep the System temperature  
// in_lrPar1 to in_lrPar2 lower than the detector temperature.
// 
// in_lrPar1  - Delta [K] to turn the heater ON:  IF L < D - in_lrPar1
// in_lrPar2  - Delta [K] to turn the heater OFF: IF L > D - in_lrPar2
//
// in_lrDelta1 > in_lrDelta2, e.g. 10K > 4K.
//
// For example:
// 	in_lrPar1 = 10K
// 	in_lrPar1 = 4K
// 	Detector temperature D = 100K
// 	The lowest system temperature is kept in range [(100-10)..(100-4)] = [90K..96K].
//	The heater is turned ON  at < 90K.
//	The heater is turned OFF at > 96K.
//
IF	stat.nState = E_CRYO_BIN_CTRL_STATE.ACTIVE_OFF  OR  
	stat.nState = E_CRYO_BIN_CTRL_STATE.ACTIVE_ON THEN
	
	IF in_lrTemp1 < in_lrTemp2 - in_lrDelta_Low THEN
		// Activate the actuator
		M_User_SetAction	:= E_CRYO_BIN_CTRL_ACTION.ON;
	ELSIF in_lrTemp1 > in_lrTemp2 - in_lrDelta_High THEN
		// Dectivate the actuator
		M_User_SetAction	:= E_CRYO_BIN_CTRL_ACTION.OFF;
	END_IF

ELSE
	// Don't do anything
	M_User_SetAction	:= E_CRYO_BIN_CTRL_ACTION.NONE;
END_IF
END_METHOD

END_FUNCTION_BLOCK

// ---- POUs/Actuators/FB_CRYO_CCC_CTRL.TcPOU
FUNCTION_BLOCK FB_CRYO_CCC_CTRL EXTENDS FB_CRYO_BIN_CTRL
VAR_INPUT
END_VAR
VAR_OUTPUT
END_VAR
VAR
	// Feedback from CCC
	{attribute 'OPC.UA.DA' := '0'}
	i_bOn				AT%I*:	BOOL;
	{attribute 'OPC.UA.DA' := '0'}
	i_bOverTemperature	AT%I*:	BOOL;
	{attribute 'OPC.UA.DA' := '0'}
	i_bUnderPressure	AT%I*:	BOOL;
END_VAR

// Set generic error if temperature inputs are not valid
IF i_bOn  AND  (i_bOverTemperature OR i_bUnderPressure) THEN
	stat.bCtrlOK	:= FALSE;
ELSE
	stat.bCtrlOK	:= TRUE;
END_IF

// Execute parent FB.
SUPER^();

METHOD M_User_SetAction : INT
VAR_INPUT
END_VAR
// TODO USER
//
// This method implements the logic for controlling a CCC.
//
// If the controller is Enabled, it should be ACTIVE_ON.
// If the controller is NOT Enabled, it should be OFF.
// 
//
IF	in_bEnable THEN
	M_User_SetAction	:= E_CRYO_BIN_CTRL_ACTION.ON;
ELSE
	M_User_SetAction	:= E_CRYO_BIN_CTRL_ACTION.OFF;
END_IF
END_METHOD

END_FUNCTION_BLOCK

// ---- POUs/Coolers/FB_CRYO_CPA.TcPOU
FUNCTION_BLOCK FB_CRYO_CPA EXTENDS FB_RS_BASE
VAR_INPUT
	{attribute 'OPC.UA.DA' := '0'}
	in_sSN_Compressor:	STRING;	// e.g. 'CPA289C-W2EHCE-180201A'
	{attribute 'OPC.UA.DA' := '0'}
	in_sSN_PulseTube:	STRING;	// e.g. 'CH40810-180208A'
	{attribute 'OPC.UA.DA' := '0'}
	in_nYear_Compressor:	INT;	// e.g. 2018
	{attribute 'OPC.UA.DA' := '0'}
	in_nYear_PulseTube:		INT;	// e.g. 2018
	{attribute 'OPC.UA.DA' := '0'}
	in_lrNextService_Compressor:	LREAL;	// Next service in absolute hours
	{attribute 'OPC.UA.DA' := '0'}
	in_lrNextService_PulseTube:		LREAL;	// Next service in absolute hours
	{attribute 'OPC.UA.DA' := '0'}
	in_nSlaveID:	BYTE := 1;		// Modbus Slave ID
	{attribute 'OPC.UA.DA' := '0'}
	in_nPeriod:		DINT := 5000;	//Interval for periodic reading [ms], default 5000 ms = 5 sec
END_VAR
VAR_OUTPUT
END_VAR
VAR CONSTANT
END_VAR
VAR
	{attribute 'OPC.UA.DA' := '1'}
	cfg:		T_CRYO_CPA_CFG;					//  Config parameters
	{attribute 'OPC.UA.DA' := '1'}
	ctrl:		T_CRYO_CPA_CTRL;				//  Control parameters
	{attribute 'OPC.UA.DA' := '1'}
	{attribute 'OPC.UA.DA.Access' := '1'}
	info:		T_CRYO_CPA_INFO; 				//  Info parameters - ReadOnly
	{attribute 'OPC.UA.DA' := '1'}
	{attribute 'OPC.UA.DA.Access' := '1'}
	stat:		T_CRYO_CPA_STAT;				//  Status parameters - ReadOnly

	{attribute 'OPC.UA.DA' := '0'}
	comm:		FB_MODBUS_COMM_CPA;				// Instance of generic comm object. OPC UA Disabled!!!
	
	(* Pointers *)
	{attribute 'OPC.UA.DA' := '0'}
	ptrCommCtrl:	POINTER TO T_MODBUS_CTRL 	:= ADR(comm.ctrl);	(* Pointer to comm.ctrl instance *)

	// I/O
	q_bCtrlStart	AT %Q*:	BOOL;	// Start control signal
	
	
	(* Timers *)
	{attribute 'OPC.UA.DA' := '0'}
	fbTimer:			TON; (* General Timeout *)
	
	// Dummy variables for testing
	nDummyWarnings:	DINT := 0;
	nDummyErrors:	DINT := 0;

END_VAR

// Set references
cfgRef	REF=cfg;
ctrlRef	REF=ctrl;
statRef	REF=stat;


// 
// Execute comm instance.
// Function 4 is used for READ.
//
comm(	in_bSimulation		:= in_bSimulation,
		in_cReadFunction	:= 4);


// Execute the base class object FB_RS_BASE
SUPER^();

METHOD ActivityInitializing
VAR_INPUT
	bExecute:	BOOL;
END_VAR
VAR_INST
	{attribute 'OPC.UA.DA' := '0'}
    nMethodState:	INT := 0;	// State Machine current state
END_VAR
VAR
	nInt:	INT;	// Temporary INT for conversion of ENUM types
END_VAR
SetAction('ActivityInitializing');


IF NOT bExecute THEN
	nMethodState	:= 0;	// Reset the state machine
	RETURN;
END_IF

// Handle State Machine
CASE nMethodState OF
	0:	// Set monitoring period (from input parameter)
		cfg.tDelay_Periodic	:= DINT_TO_TIME(in_nPeriod);
		// Auto monitor, i.e. monitor in Standby_Ready as well
		cfg.bAutoMonitor	:= TRUE;

		(* Set initial state and status *)
		stat.bInitialised	:= FALSE;
		stat.nRetries		:= 0;

		SetStatus(E_SM_ERROR.OK, 'BUSY');
		
		// User configuration of the system
		M_UserConfigure();

		nMethodState := 10;				// Go to next state, i.e. INIT_COMM

	10:	// Initialize COMM port, i.e. Reset the serial port.
		nInt	:= E_RS_COMM_CMD.INIT;
		ptrCommCtrl^.nCommand	:= nInt;
		ptrCommCtrl^.bExecute	:= TRUE;

		(* Start the timer by going false/true *)
		fbTimer (IN := FALSE); (* Reset timer *)
		fbTimer (IN := TRUE, PT := T#5S); (* 5 sec timeout for reply *)

		nMethodState := 15;	// On next cycle wait until comm port is reset, i.e. idle
		
	15:	// Wait IDLE or ERROR
		fbTimer (IN := TRUE);
		IF comm.stat.nStatus = E_RS_COMM_STATUS.IDLE THEN
			// Communication is IDLE 
			fbTimer (IN := FALSE);	// disable timer 
			stat.nInputBuffer		:= comm.stat.DeviceReply;	// Save the reply

			bCommProblem	:= FALSE;
			// Device INIT is done.
			// INITDONE will bring it to OPERATIONAL
			stat.bInitialised 	:= TRUE;
			SetStatus(E_CCC_STATUS.IDLE, 'IDLE');
			nEvent 	:= E_SM_EVENT.INITDONE;
			RETURN;
		ELSIF comm.stat.nStatus = E_RS_COMM_STATUS.ERROR OR fbTimer.Q THEN
			// There is an error.
			// Re-initialise the comm port.
			// This is the only thing we can do.
			SetStatus(E_CCC_ERROR.COMM, 'ERROR: Communication error');	
			bCommProblem	:= TRUE;
			nMethodState	:= 10;		// Retry to INIT_COMM
			RETURN;
		END_IF
	
END_CASE
END_METHOD

METHOD ActivityMonitoring
VAR_INPUT
	bExecute:	BOOL;
END_VAR
VAR_INST
	{attribute 'OPC.UA.DA' := '0'}
    nMethodState:	INT := 0;					// State Machine current state
	{attribute 'OPC.UA.DA' := '0'}
	nSlaveIndex:	INT := 1;
	{attribute 'OPC.UA.DA' := '0'}
	nRetries:		INT := 0;					// Number of retries in case of communication problems
END_VAR
IF NOT bExecute THEN
	SetAction('ActivityMonitoring'); 
	SetStatus(E_SM_ERROR.OK, 'BUSY');
	nMethodState	:= 0;	// Reset the state machine
	ctrl.nSlaveID	:= cfg.nSlaveID;
	ctrl.nRegister	:= cfg.nAddrCommon;
	ctrl.nWords		:= cfg.nWordsCommon;
	nRetries		:= 0;					
	RETURN;
END_IF

// Handle State Machine
CASE nMethodState OF
	0:	// Execute a command from the command array
		// Check if we have to exit Monitoring
		
		// Send command
		ptrCommCtrl^.nCommand	:= E_MODBUS_CMD.SEND;
		ptrCommCtrl^.nSlaveID	:= ctrl.nSlaveID;
		ptrCommCtrl^.nRegister	:= ctrl.nRegister;
		ptrCommCtrl^.nWords		:= ctrl.nWords;
		ptrCommCtrl^.bExecute	:= TRUE;
		
		(* Start the timer by going false/true *)
		fbTimer (IN := FALSE); (* Reset timer *)
		fbTimer (IN := TRUE, PT := T#5S); (* 5 sec timeout for reply *)

		nMethodState := 20;				// Goto WAIT for Reading to complete,

	10:	// Wait until the delay timeout expires
		fbTimer (IN := TRUE);

		(* If Timer has expired, go to the next state. *)
		IF fbTimer.Q THEN
			fbTimer (IN := FALSE);
			SetStatus(E_SM_ERROR.OK, 'BUSY');
			nMethodState 	:= 0;	// Goto next reading
			RETURN;
		END_IF
	


	20:	// Wait for the reading to complete, i.e. IDLE
		fbTimer (IN := TRUE);
		IF comm.stat.nStatus = E_RS_COMM_STATUS.IDLE THEN
			//
			// Communication is IDLE. Everything is fine. 
			//
			fbTimer (IN := FALSE);	// disable timer 
			stat.nInputBuffer	:= comm.stat.DeviceReply;	// Save the reply
			
			//
			// Extract the readings from the reply.
			//
			M_ExtractReadings();
			
			bCommProblem	:= FALSE;
			nRetries		:= 0;	// Reset number of retries
			
			// Wait tDelay_Periodic before re-starting the READ.
			SetStatus(E_SM_ERROR.OK, 'IDLE');
			(* Start the timer by going false/true *)
			fbTimer (IN := FALSE); (* Reset timer *)
			fbTimer (IN := TRUE, PT := cfg.tDelay_Periodic);
			nMethodState := 10;				// Goto Wait 
			RETURN;

		ELSIF INT_TO_DINT(comm.stat.nStatus) = INT_TO_DINT(E_MODBUS_STATUS.ERROR) OR fbTimer.Q THEN
			//
			// There is a communication problem. 
			// Re-initialise comm port.
			//
			fbTimer (IN := FALSE);
			SetStatus(E_MODBUS_ERROR.RECEIVE, 'ERROR: Communication error');	
			bCommProblem	:= TRUE;
			
			// Keep track of how many times we re-tried
			nRetries		:= nRetries + 1;		// Increment number of retries
			stat.nRetries	:= stat.nRetries + 1;	// Increment total number of retries

			// Re-initialise the comm port
			ptrCommCtrl^.nCommand	:= E_MODBUS_CMD.INIT;
			ptrCommCtrl^.bExecute	:= TRUE;
			// Apply a delay of 3 sec and retry
			fbTimer (IN := FALSE); (* Reset timer *)
			fbTimer (IN := TRUE, PT := T#3000MS);
			nMethodState := 10;				// Goto Wait 
			RETURN;
		END_IF

	
END_CASE
END_METHOD

METHOD CheckForEvents
VAR_INPUT
END_VAR
VAR
//	nInt2:	INT;	// Temporary INT for conversion of ENUM types
END_VAR

(* 
	Check for events in the following order: 
   	1) HW failure: without HW avilability there is no point to do anything
	2) Internal events: to allow completing the initiated commands before 
                        starting processing new commands. 
   	3) Commands: to react to external commands. Commands should be executed 
                 before processing HW signals to allow to start a recovery action.
   	4) HW signals: if any.
*)

IF NOT M_GetCouplerState() THEN	
	(* Check if the HW is NOT OK *)
	(*
	If the hardware status is NOT OK, we cannot trust the readings.
	Variable i_nCouplerState has to be mapped to a State of a terminal, e.g. EK1100.
	The value should be 8.
 	*)
	SetEvent(E_SM_EVENT.ERRHW);
	SetStatus(E_SM_ERROR.HW_NOT_OP, 'ERROR: HW not in OPERATIONAL state');

ELSIF ctrlRef.bExecute  THEN
	// Check for CPA specific commands.
	// TODO SetLastCommand() and SetEvent() don't work here. Check it!!!
	ctrlRef.bExecute	:= FALSE;			(* Clear the Execute bit *)
	SetLastCommand(E_RS_COMMAND.CTRL_CMD);	// Save the last command
	SetEvent(E_RS_COMMAND.CTRL_CMD);
	IF	ctrl.nDevCommand = E_CRYO_CPA_CMDS.START	THEN
		// Set control signal to TRUE.
		// This will start the compressor.
		q_bCtrlStart	:= TRUE;
	ELSIF	ctrl.nDevCommand = E_CRYO_CPA_CMDS.STOP	THEN
		// Set control signal to FALSE.
		// This will stop the compressor.
		q_bCtrlStart	:= FALSE;
	ELSE
		(* Handle standard RS commands *)
		SetLastCommand(ctrlRef.nCommand);			(* Save the last command *)
		SetEvent(ctrlRef.nCommand);
	END_IF
	ctrlRef.bExecute	:= FALSE;			(* Clear the Execute bit *)
	ctrlRef.nCommand 	:= E_RS_COMMAND.NONE;	(* Clear the Command *)
ELSIF nInternalEvent <> E_SM_EVENT.NONE THEN
	(* Handle internal events *)
	SetEvent(nInternalEvent);
	nInternalEvent := E_SM_EVENT.NONE;
ELSE
	(* Handle HW problems and unexpected bahaviour *)
	
END_IF
END_METHOD

METHOD M_ByteSwapFLOAT : LREAL
VAR_INPUT
	pByte:		POINTER TO BYTE;	// Pointer to array of bytes read from JUMO
END_VAR
VAR
	rResult:	REAL;
	pResult:	POINTER TO BYTE	:= ADR(rResult);	// Pointer to the result
END_VAR
pResult[0]	:= pByte[1];
pResult[1]	:= pByte[0];
pResult[2]	:= pByte[3];
pResult[3]	:= pByte[2];

M_ByteSwapFLOAT	:= REAL_TO_LREAL(rResult);
END_METHOD

METHOD M_ByteSwapINT : INT
VAR_INPUT
	pByte:		POINTER TO BYTE;	// Pointer to array of bytes read from JUMO
END_VAR
VAR
	nResult:	INT;
	pResult:	POINTER TO BYTE	:= ADR(nResult);	// Pointer to the result
END_VAR
pResult[0]	:= pByte[1];
pResult[1]	:= pByte[0];

M_ByteSwapINT	:= nResult;
END_METHOD

METHOD M_CheckDiagnostics
VAR_INPUT
END_VAR
VAR
	nTmp:		DINT;
	i:			INT;
	sTmp:		STRING(56) := '';
END_VAR
// Process warnings/alarms
//M_CheckWarnings(stat.lrWarningState);
M_CheckWarnings(nDummyWarnings);

// Process errors
//M_CheckErrors(stat.lrWarningState);
M_CheckErrors(nDummyErrors);
END_METHOD

METHOD M_CheckErrors
VAR_INPUT
	nErrors:	DINT;
END_VAR
VAR
	nTmp:		UDINT;
	nRef:		UDINT	:= 16#00000001;
	bProblem:	BOOL	:= FALSE;
	i:			INT;
END_VAR
nTmp	:= DINT_TO_UDINT(-nErrors);


FOR i := 0 TO 6 DO
	// Check for 'too low' errors
	IF		(stat.aReadings[i] < cfg.aLimits[i].rErrorLow) OR
			((nTmp AND SHL(nRef,cfg.aDiag[i].nBitLow)) <> 0)	THEN
		bProblem	:= TRUE;
		stat.arrErrors[i]		:= E_CRYO_CPA_ALARM.LOW;
		M_SetAlarmText(i);	// Error string for going low
	// Check for 'too high' errors
	ELSIF	(stat.aReadings[i] > cfg.aLimits[i].rErrorHigh) OR
			((nTmp AND SHL(nRef,cfg.aDiag[i].nBitHigh)) <> 0)	THEN
		bProblem	:= TRUE;
		stat.arrErrors[i]		:= E_CRYO_CPA_ALARM.HIGH;
		M_SetAlarmText(i);	// Error string for going high
	ELSE
		stat.arrErrors[i]	:= E_CRYO_CPA_ALARM.NONE;
	END_IF
END_FOR

// Check if there are any errors.
IF NOT bProblem THEN
	// No error. Clear all and write OK in warning text.
	FOR i := 0 TO 6 DO
		stat.arrErrors[i]	:= E_CRYO_CPA_ALARM.NONE;
	END_FOR
	stat.sError := '';
//  We don't touch stat.nStatusCode! It might have been set with alarm.
	RETURN;
ELSE
	stat.nStatusCode	:= 2;	// Error
END_IF
END_METHOD

METHOD M_CheckService
VAR_INPUT
END_VAR
VAR
    fbFormat: FB_FormatString;
	lrHoursLeft:	LREAL;
END_VAR
//
// Check compressor hours
//
lrHoursLeft	:= in_lrNextService_Compressor - stat.lrHoursOfOperation;
IF lrHoursLeft < cfg.lrServiceDue_Compressor THEN
	stat.bServiceDue_Compressor	:= TRUE;
	stat.wColour_Compressor		:= 16#FFFF0000;
	IF lrHoursLeft >= 0.0 THEN
		fbFormat( 	sFormat := 'Service due in %.0f hours', 
					arg1 := F_LREAL( lrHoursLeft ), 
					sOut => stat.sServiceDue_Compressor);
	ELSE
		lrHoursLeft	:= -1 * lrHoursLeft;
		fbFormat( 	sFormat := 'Service overdue by %.0f hours', 
					arg1 := F_LREAL( lrHoursLeft ), 
					sOut => stat.sServiceDue_Compressor);
	END_IF
ELSE
	stat.wColour_Compressor		:= 16#FF0000FF;
	stat.bServiceDue_Compressor	:= FALSE;
	stat.sServiceDue_Compressor	:= 'OK';
END_IF

//
// Check pulse tube hours
//
lrHoursLeft	:= in_lrNextService_PulseTube - stat.lrHoursOfOperation;
IF lrHoursLeft < cfg.lrServiceDue_PulseTube THEN
	stat.bServiceDue_PulseTube	:= TRUE;
	stat.wColour_PulseTube		:= 16#FFFF0000;
	IF lrHoursLeft >= 0.0 THEN
		fbFormat( 	sFormat := 'Service due in %.0f hours', 
					arg1 := F_LREAL( lrHoursLeft ), 
					sOut => stat.sServiceDue_PulseTube);
	ELSE
		lrHoursLeft	:= -1 * lrHoursLeft;
		fbFormat( 	sFormat := 'Service overdue by %.0f hours', 
					arg1 := F_LREAL( lrHoursLeft ), 
					sOut => stat.sServiceDue_PulseTube);
	END_IF
ELSE
	stat.wColour_PulseTube		:= 16#FF0000FF;
	stat.bServiceDue_PulseTube	:= FALSE;
	stat.sServiceDue_PulseTube	:= 'OK';
END_IF
END_METHOD

METHOD M_CheckWarnings
VAR_INPUT
	nWarnings:	DINT;
END_VAR
VAR
	nTmp:		UDINT;
	nRef:		UDINT	:= 16#00000001;
	bProblem:	BOOL	:= FALSE;
	i:			INT;
END_VAR
// Warning are given as negative numbers.
// Change the sign and then do checks with bit shifts to the left.
nTmp	:= DINT_TO_UDINT(-nWarnings);

// Check warnings one by one
FOR i := 0 TO 6 DO
	// Check for 'running low' warnings/alarms
	IF		(stat.aReadings[i] < cfg.aLimits[i].rAlarmLow) OR
			((nTmp AND SHL(nRef,cfg.aDiag[i].nBitLow)) <> 0)	THEN
		bProblem	:= TRUE;
		stat.arrAlarms[i]		:= E_CRYO_CPA_ALARM.LOW;
		M_SetAlarmText(i);	// Alarm string for going low (FALSE)
	// Check for 'running high' warnings/alarms
	ELSIF	(stat.aReadings[i] > cfg.aLimits[i].rAlarmHigh) OR
			((nTmp AND SHL(nRef,cfg.aDiag[i].nBitHigh)) <> 0)		THEN
		bProblem	:= TRUE;
		stat.arrAlarms[i]		:= E_CRYO_CPA_ALARM.HIGH;
		M_SetAlarmText(i);	// Alarm string for going high (TRUE)
	ELSE
		stat.arrAlarms[i]	:= E_CRYO_CPA_ALARM.NONE;
	END_IF
END_FOR

// Check if there are any alarms.
IF NOT bProblem THEN
	// No alarms. Clear all and write OK in warning text.
	FOR i := 0 TO 6 DO
		stat.arrAlarms[i]	:= E_CRYO_CPA_ALARM.NONE;
	END_FOR
	stat.sAlarm := '';
	stat.nStatusCode	:= 0;	// OK
ELSE
	stat.nStatusCode	:= 1;	// Alarm
END_IF
END_METHOD

METHOD M_ExtractReadings : BOOL
VAR_INPUT
END_VAR
VAR
	pBuf:	POINTER TO BYTE	:= ADR(stat.nInputBuffer);
	nPos:	INT	:= 0;	// byte position in the buffer
	pPtr:	POINTER TO UINT;	// Pointer to the result
END_VAR
// There are 3 bytes before data starts !!!
////////////////////////////
// Extract Common Parameters
// Buffer starts from 30,001
// 3 bytes before real data
////////////////////////////

// nOperatingState
// 30,001 - Operating State
// Offset 3 + 0x2 = 3
nPos	:= cfg.nPosOffset + 3;
stat.nOperatingState := M_ByteSwapINT(ADR(pBuf[nPos]));

// nCompressorRunning
// 30,002 - Compressor Running
// Offset 3 + 1x2 = 5
nPos	:= nPos + 2;
stat.nCompressorRunning := M_ByteSwapINT(ADR(pBuf[nPos]));

// 
// 
// Offset 3 + x2 = 
nPos	:= nPos + 2;
stat.lrWarningState := M_ByteSwapFLOAT(ADR(pBuf[nPos]));

// 
// 
// Offset 3 + x2 = 
nPos	:= nPos + 4;
stat.lrAlarmState := M_ByteSwapFLOAT(ADR(pBuf[nPos]));

// lrCoolantInTemp
// 30,007 - Coolant In Temp
// Offset 3 + 6x2 = 15
nPos	:= nPos + 4;
stat.lrCoolantInTemp	:= M_ByteSwapFLOAT(ADR(pBuf[nPos]));

// lrCoolantOutTemp
// 30,009 - Coolant Out Temp
// Offset 3 + 8x2 = 19
nPos	:= nPos + 4;
stat.lrCoolantOutTemp	:= M_ByteSwapFLOAT(ADR(pBuf[nPos]));

// lrOilTemp
// 30,011 - Oil Temp
// Offset 3 + 10x2 = 23
nPos	:= nPos + 4;
stat.lrOilTemp	:= M_ByteSwapFLOAT(ADR(pBuf[nPos]));

nPos	:= nPos + 4;
stat.lrHeliumTemp	:= M_ByteSwapFLOAT(ADR(pBuf[nPos]));

nPos	:= nPos + 4;
stat.lrLowPressure	:= M_ByteSwapFLOAT(ADR(pBuf[nPos]));

nPos	:= nPos + 4;
stat.lrLowPressureAverage	:= M_ByteSwapFLOAT(ADR(pBuf[nPos]));

nPos	:= nPos + 4;
stat.lrHighPressure	:= M_ByteSwapFLOAT(ADR(pBuf[nPos]));

nPos	:= nPos + 4;
stat.lrHighPressureAverage	:= M_ByteSwapFLOAT(ADR(pBuf[nPos]));

nPos	:= nPos + 4;
stat.lrDeltaPressureAverage	:= M_ByteSwapFLOAT(ADR(pBuf[nPos]));

nPos	:= nPos + 4;
stat.lrMotorCurrent	:= M_ByteSwapFLOAT(ADR(pBuf[nPos]));

nPos	:= nPos + 4;
stat.lrHoursOfOperation	:= M_ByteSwapFLOAT(ADR(pBuf[nPos]));

nPos	:= nPos + 4;
stat.nPressureScale	:= M_ByteSwapINT(ADR(pBuf[nPos]));

nPos	:= nPos + 2;
stat.nTempScale	:= M_ByteSwapINT(ADR(pBuf[nPos]));

nPos	:= nPos + 2;
pPtr	:= ADR(pBuf[nPos]);
stat.nPanelSerialNumber	:= pPtr^;
//stat.nPanelSerialNumber	:= M_ByteSwapINT(ADR(pBuf[nPos]));

nPos	:= nPos + 2;
stat.nModelMajorMinor	:= M_ByteSwapINT(ADR(pBuf[nPos]));

//////////////////////////
// Assign values to arrays
//////////////////////////

stat.aReadings[E_CRYO_CPA_DIAG_IDX.WATER_IN]	:= stat.lrCoolantInTemp;
stat.aReadings[E_CRYO_CPA_DIAG_IDX.WATER_OUT]	:= stat.lrCoolantOutTemp;
stat.aReadings[E_CRYO_CPA_DIAG_IDX.OIL_TEMP]	:= stat.lrOilTemp;
stat.aReadings[E_CRYO_CPA_DIAG_IDX.HELIUM_TEMP]	:= stat.lrHeliumTemp;
stat.aReadings[E_CRYO_CPA_DIAG_IDX.HELIUM_LOW_PRESS_OP]		:= stat.lrLowPressure;
stat.aReadings[E_CRYO_CPA_DIAG_IDX.HELIUM_HIGH_PRESS_OP]	:= stat.lrHighPressure;

IF stat.nCompressorRunning <> 0 THEN
	stat.bSystemOn	:= TRUE;
	cfg.aLimits	:= cfg.aLimits_OP;
	
	// System is ON. Set 'operational' values to the actual reading.
	stat.aReadings[E_CRYO_CPA_DIAG_IDX.HELIUM_DELTA_PRESS]		:= stat.lrDeltaPressureAverage;
ELSE
	stat.bSystemOn	:= FALSE;
	cfg.aLimits	:= cfg.aLimits_ST;
	
	// System is OFF. 
	// Set 'static' values to the middle of the valid range to avoid warnings and errors.
	stat.aReadings[E_CRYO_CPA_DIAG_IDX.HELIUM_DELTA_PRESS]		:= 12.0;	// dummy
END_IF

//
// Check for Alarms and Errors
//
M_CheckDiagnostics();

//
// Get Model Number
//
M_GetModelNumber();

//
// Get Operational State
//
M_GetOperatingState();

//
// Check due service
//
M_CheckService();
END_METHOD

METHOD M_GetModelNumber
VAR_INPUT
END_VAR
VAR
	nModelMajor:	SINT;
	nModelMinor:	SINT;
	nVersionMajor:	SINT;
	nVersionMinor:	SINT;
	pPtr:			POINTER TO BYTE;;	// Pointer to the result
	sModelMajor, sModelMinor:	STRING(16);
	sVersionMajor, sVersionMinor:	STRING(16);
	sTmp:	STRING;
END_VAR
// Get major and minor version of the model
pPtr	:= ADR(stat.nModelMajorMinor);
nModelMinor	:= BYTE_TO_SINT(pPtr^);

pPtr	:= ADR(stat.nModelMajorMinor) + 1;
nModelMajor	:= BYTE_TO_SINT(pPtr^);

CASE nModelMajor OF
	1:	sModelMajor	:= '8';
	2:	sModelMajor	:= '9';
	3:	sModelMajor	:= '10';
	4:	sModelMajor	:= '11';
	5:	sModelMajor	:= '28';
END_CASE

CASE nModelMinor OF
	1:	sModelMinor	:= 'A1';
	2:	sModelMinor	:= '01';
	3:	sModelMinor	:= '02';
	4:	sModelMinor	:= '03';
	5:	sModelMinor	:= 'H3';
	6:	sModelMinor	:= 'I3';
	7:	sModelMinor	:= '04';
	8:	sModelMinor	:= 'H4';
	9:	sModelMinor	:= '05';
	10:	sModelMinor	:= 'H5';
	11:	sModelMinor	:= 'I6';
	12:	sModelMinor	:= '06';
	13:	sModelMinor	:= '07';
	14:	sModelMinor	:= 'H7';
	15:	sModelMinor	:= 'I7';
	16:	sModelMinor	:= '08';
	17:	sModelMinor	:= '09';
	18:	sModelMinor	:= '9C';
	19:	sModelMinor	:= '10';
	20:	sModelMinor	:= '1I';
	21:	sModelMinor	:= '11';
	22:	sModelMinor	:= '12';
	23:	sModelMinor	:= '13';
	24:	sModelMinor	:= '14';
END_CASE

// Get major and minor version of the panel
pPtr	:= ADR(stat.nPanelSerialNumber);
nVersionMinor	:= BYTE_TO_SINT(pPtr^);

pPtr	:= ADR(stat.nPanelSerialNumber) + 1;
nVersionMajor	:= BYTE_TO_SINT(pPtr^);


sTmp	:= 'CRYOMECH CPA';
sTmp	:= concat(concat(sTmp,sModelMajor),sModelMinor);
sTmp	:= concat(concat(sTmp,'   ID: '),in_sName);
//sTmp	:= concat(concat(sTmp,'.'),SINT_TO_STRING(nVersionMinor));

stat.sModelNumber	:= sTmp;



(*
Major Model Numbers consist of
1: 800 Series
2: 900 Series
3: 1000 Series
4: 1100 Series
5: 2800 Series
Minor Model Numbers consist of:
1: A1 13: 07
2: 01 14: H7
3: 02 15: I7
4: 03 16: 08
5: H3 17: 09
6: I3 18: 9C
7: 04 19: 10
8: H4 20: 1I
9: 05 21: 11
10: H5 22: 12
11: I6 23: 13
12: 06 24: 14
*)
END_METHOD

METHOD M_GetOperatingState
VAR_INPUT
END_VAR

VAR
	
END_VAR
CASE stat.nOperatingState OF
	0: stat.sOperatingState := 'Idling - ready to start';
	2: stat.sOperatingState := 'Starting';
	3: stat.sOperatingState := 'Running';
	5: stat.sOperatingState := 'Stopping';
	6: stat.sOperatingState := 'Error Lockout';
	7: stat.sOperatingState := 'Error';
	8: stat.sOperatingState := 'Helium Cool Down';
	9: stat.sOperatingState := 'Error-Power Related';
	16: stat.sOperatingState := 'Error Recovery';
END_CASE




(*
Input Register 30001: (operating state)
0: Idling - ready to start
2: Starting
3: Running
5: Stopping
6: Error Lockout
7: Error
8: Helium Cool Down
9: Error-Power Related
16: Error Recovery
*)
END_METHOD

METHOD M_SetAlarmText
VAR_INPUT
	nIndex:	INT;	// alarm index
END_VAR
VAR
	sTmp1:	STRING(128);
END_VAR
//
// Handle alarms
//
IF stat.arrAlarms[nIndex] = E_CRYO_CPA_ALARM.NONE THEN
	// No alarm 
	stat.sAlarm	:= '';
ELSIF stat.arrAlarms[nIndex] = E_CRYO_CPA_ALARM.LOW THEN
	// Alarm text, e.g. 
	// ‘Alarm: High pressure running low, compressor will shut off at 27.6 bar’
	sTmp1	:= concat('Alarm: ', cfg.aDiag[nIndex].sLabel);
	sTmp1	:= concat(sTmp1, ' running low. It will shut down at ');
	sTmp1	:= concat(sTmp1, LREAL_TO_STRING(cfg.aDiag[nIndex].rErrorLow));
	sTmp1	:= concat(sTmp1, concat(' ', cfg.aDiag[nIndex].sUnits));
	stat.sAlarm	:= sTmp1;
ELSIF stat.arrAlarms[nIndex] = E_CRYO_CPA_ALARM.HIGH THEN
	// Alarm text, e.g. 
	// ‘Alarm: High pressure running high, compressor will shut off at 27.6 bar’
	sTmp1	:= concat('Alarm: ', cfg.aDiag[nIndex].sLabel);
	sTmp1	:= concat(sTmp1, ' running high. It will shut down at ');
	sTmp1	:= concat(sTmp1, LREAL_TO_STRING(cfg.aDiag[nIndex].rErrorHigh));
	sTmp1	:= concat(sTmp1, concat(' ', cfg.aDiag[nIndex].sUnits));
	stat.sAlarm	:= sTmp1;
END_IF

//
// Handle errors
//
IF stat.arrErrors[nIndex] = E_CRYO_CPA_ALARM.NONE THEN
	// No error 
	stat.sError	:= '';
ELSIF stat.arrErrors[nIndex] = E_CRYO_CPA_ALARM.LOW THEN
	// Error text, e.g. 
	// ‘Error: High pressure was too low, compressor shut down at 27.6 bar’
	sTmp1	:= concat('Error: ', cfg.aDiag[nIndex].sLabel);
	sTmp1	:= concat(sTmp1, ' was too low. Shutdown was at ');
	sTmp1	:= concat(sTmp1, LREAL_TO_STRING(cfg.aDiag[nIndex].rErrorLow));
	sTmp1	:= concat(sTmp1, concat(' ', cfg.aDiag[nIndex].sUnits));
	stat.sError	:= sTmp1;
ELSIF stat.arrErrors[nIndex] = E_CRYO_CPA_ALARM.HIGH THEN
	// Error text, e.g. 
	// ‘Error: High pressure was too high, compressor shut down at 27.6 bar’
	sTmp1	:= concat('Error: ', cfg.aDiag[nIndex].sLabel);
	sTmp1	:= concat(sTmp1, ' was too high. Shutdown was at ');
	sTmp1	:= concat(sTmp1, LREAL_TO_STRING(cfg.aDiag[nIndex].rErrorHigh));
	sTmp1	:= concat(sTmp1, concat(' ', cfg.aDiag[nIndex].sUnits));
	stat.sError	:= sTmp1;
END_IF
END_METHOD

METHOD M_UserConfigure : BOOL
VAR_INPUT
END_VAR
VAR
	i, j:	int;
END_VAR
// TODO USER
// Add here real configuration

// SlaveID
cfg.nSlaveID	:= in_nSlaveID;

// We always read from CPA
ctrl.nCmdType	:= E_MODBUS_CMD_TYPE.READ;

ctrl.nRegister	:= cfg.nAddrCommon;
ctrl.nWords		:= cfg.nWordsCommon;

//
// Configure OP and STATIC limits
FOR i := 0 TO 6 DO
	cfg.aLimits_OP[i].rAlarmLow	:= MAX(cfg.aDiag[i].rAlarmLow_CPA,  cfg.aDiag[i].rAlarmLow_ESO);
	cfg.aLimits_OP[i].rAlarmHigh	:= MIN(cfg.aDiag[i].rAlarmHigh_CPA, cfg.aDiag[i].rAlarmHigh_ESO);
	cfg.aLimits_OP[i].rErrorLow	:= cfg.aDiag[i].rErrorLow;
	cfg.aLimits_OP[i].rErrorHigh	:= cfg.aDiag[i].rErrorHigh;

	j	:= i;
	IF	i = E_CRYO_CPA_DIAG_IDX.HELIUM_LOW_PRESS_OP OR 
		i = E_CRYO_CPA_DIAG_IDX.HELIUM_HIGH_PRESS_OP THEN
		j	:= i+3;	// Use STATIC limits
	END_IF
	cfg.aLimits_ST[i].rAlarmLow	:= MAX(cfg.aDiag[j].rAlarmLow_CPA,  cfg.aDiag[j].rAlarmLow_ESO);
	cfg.aLimits_ST[i].rAlarmHigh	:= MIN(cfg.aDiag[j].rAlarmHigh_CPA, cfg.aDiag[j].rAlarmHigh_ESO);
	cfg.aLimits_ST[i].rErrorLow	:= cfg.aDiag[j].rErrorLow;
	cfg.aLimits_ST[i].rErrorHigh	:= cfg.aDiag[j].rErrorHigh;
END_FOR
END_METHOD

END_FUNCTION_BLOCK

// ---- POUs/Comm/FB_MODBUS_COMM_CPA.TcPOU
FUNCTION_BLOCK FB_MODBUS_COMM_CPA EXTENDS FB_MODBUS_COMM_BASE
VAR_INPUT
END_VAR
VAR_OUTPUT
END_VAR
VAR CONSTANT
END_VAR
VAR
	{attribute 'OPC.UA.DA' := '0'}
	sim:		FB_SIM_MODBUS_COMM_CPA;	// Reference to COMM simulator

END_VAR

simRef	REF=sim;

// Execute base FB, i.e. FB_MODBUS_COMM_BASE.
SUPER^();

END_FUNCTION_BLOCK

// ---- POUs/Simulation/FB_SIM_MODBUS_COMM_CPA.TcPOU
FUNCTION_BLOCK FB_SIM_MODBUS_COMM_CPA EXTENDS FB_SIM_MODBUS_COMM_BASE
VAR_INPUT
END_VAR
VAR_OUTPUT
END_VAR
VAR
END_VAR

M_ActivityDo();

METHOD M_GetSimReply : STRING(255)
VAR_INPUT
	{attribute 'OPC.UA.DA' := '0'}
	cmd:	STRING(16);		// MODBUS command. Only first 8 bytes are used
END_VAR
VAR
	sReply:		ARRAY [0..300] OF BYTE;
	sReply1:	STRING(255);
	n2Bytes:	ARRAY [0..1] OF BYTE;	// 2 bytes
	n4Bytes:	ARRAY [0..3] OF BYTE;	// 4 bytes
	i:			INT;
	nRegister:	INT;
	nWords:		INT;
	nPos:		INT;	
END_VAR
// TODO User: Implement simulator replies in FBs that EXTEND FB_SIM_MODBUS_COMM_BASE.
//            Only case where cmd[1] = E_MODBUS_CMD_TYPE.READ should be implemented.

IF cmd[1] = E_MODBUS_CMD_TYPE.WRITE THEN
// This is a WRITE command.
// Reply is the same as the command.
(*
	FOR i:=0 TO 8 DO
		sReply[i]	:= cmd[i];
	END_FOR
	*)
	M_GetSimReply := cmd;	
ELSE
// This is a READ command
	// Get register number - cmd[2..3] swapped bytes
	nRegister	:= M_ByteSwapINT(ADR(cmd[2]));

	// Get number of words - cmd[4..5] swapped bytes
	nWords	:= M_ByteSwapINT(ADR(cmd[4]));

	sReply[0]	:= cmd[0];
	sReply[1]	:= cmd[1];
	sReply[2]	:= INT_TO_BYTE(nWords * 2);
	
	IF nRegister = 16#0001 THEN		// common data
// nOperatingState
// 30,001 - Operating State
// 	3: stat.sOperatingState := 'Running';
// Offset 3 + 0x2 = 3
		nPos	:= 3;
		n2Bytes := M_ByteSwap_INT_TO_BYTES(3);
		M_InsertBytes_INT(s1:=sReply, s2:=n2Bytes, nPos:=nPos);

// nCompressorRunning
// 30,002 - Compressor Running == 1
// Offset 3 + 1x2 = 5
		nPos	:= 5;
		n2Bytes := M_ByteSwap_INT_TO_BYTES(1);
		M_InsertBytes_INT(s1:=sReply, s2:=n2Bytes, nPos:=nPos);

// nPos	:= nPos + 2;
// stat.lrWarningState := M_ByteSwapFLOAT(ADR(pBuf[nPos]));
		nPos	:= 7;
		n4Bytes := M_ByteSwap_REAL_TO_BYTES(0.0);
		M_InsertBytes_REAL(s1:=sReply, s2:=n4Bytes, nPos:=nPos);

// nPos	:= nPos + 4;
// stat.lrAlarmState := M_ByteSwapFLOAT(ADR(pBuf[nPos]));
		nPos	:= 11;
		n4Bytes := M_ByteSwap_REAL_TO_BYTES(0.0);
		M_InsertBytes_REAL(s1:=sReply, s2:=n4Bytes, nPos:=nPos);

// lrCoolantInTemp
// 30,007 - Coolant In Temp
// Offset 3 + 6x2 = 15
// nPos	:= nPos + 4;
// stat.lrCoolantInTemp	:= M_ByteSwapFLOAT(ADR(pBuf[nPos]));
		nPos	:= 15;
		n4Bytes := M_ByteSwap_REAL_TO_BYTES(M_GenerateRandom_REAL(17.0,1.0));
		M_InsertBytes_REAL(s1:=sReply, s2:=n4Bytes, nPos:=nPos);

// lrCoolantOutTemp
// 30,009 - Coolant Out Temp
// Offset 3 + 8x2 = 19
// nPos	:= nPos + 4;
// stat.lrCoolantOutTemp	:= M_ByteSwapFLOAT(ADR(pBuf[nPos]));
		nPos	:= 19;
		n4Bytes := M_ByteSwap_REAL_TO_BYTES(M_GenerateRandom_REAL(28.5,1.0));
		M_InsertBytes_REAL(s1:=sReply, s2:=n4Bytes, nPos:=nPos);

// lrOilTemp
// 30,011 - Oil Temp
// Offset 3 + 10x2 = 23
//nPos	:= nPos + 4;
//stat.lrOilTemp	:= M_ByteSwapFLOAT(ADR(pBuf[nPos]));
		nPos	:= 23;
		n4Bytes := M_ByteSwap_REAL_TO_BYTES(M_GenerateRandom_REAL(25.0,1.0));
		M_InsertBytes_REAL(s1:=sReply, s2:=n4Bytes, nPos:=nPos);

//nPos	:= nPos + 4;
//stat.lrHeliumTemp	:= M_ByteSwapFLOAT(ADR(pBuf[nPos]));
		nPos	:= 27;
		n4Bytes := M_ByteSwap_REAL_TO_BYTES(M_GenerateRandom_REAL(42.0,1.0));
		M_InsertBytes_REAL(s1:=sReply, s2:=n4Bytes, nPos:=nPos);


//nPos	:= nPos + 4;
//stat.lrLowPressure	:= M_ByteSwapFLOAT(ADR(pBuf[nPos]));
		nPos	:= 31;
		n4Bytes := M_ByteSwap_REAL_TO_BYTES(M_GenerateRandom_REAL(8.5,1.0));
		M_InsertBytes_REAL(s1:=sReply, s2:=n4Bytes, nPos:=nPos);

//nPos	:= nPos + 4;
//stat.lrLowPressureAverage	:= M_ByteSwapFLOAT(ADR(pBuf[nPos]));
		nPos	:= 35;
		n4Bytes := M_ByteSwap_REAL_TO_BYTES(M_GenerateRandom_REAL(8.5,1.0));
		M_InsertBytes_REAL(s1:=sReply, s2:=n4Bytes, nPos:=nPos);

//nPos	:= nPos + 4;
//stat.lrHighPressure	:= M_ByteSwapFLOAT(ADR(pBuf[nPos]));
		nPos	:= 39;
		n4Bytes := M_ByteSwap_REAL_TO_BYTES(M_GenerateRandom_REAL(21.0,1.0));
		M_InsertBytes_REAL(s1:=sReply, s2:=n4Bytes, nPos:=nPos);

//nPos	:= nPos + 4;
//stat.lrHighPressureAverage	:= M_ByteSwapFLOAT(ADR(pBuf[nPos]));
		nPos	:= 43;
		n4Bytes := M_ByteSwap_REAL_TO_BYTES(M_GenerateRandom_REAL(21.0,1.0));
		M_InsertBytes_REAL(s1:=sReply, s2:=n4Bytes, nPos:=nPos);

//nPos	:= nPos + 4;
//stat.lrDeltaPressureAverage	:= M_ByteSwapFLOAT(ADR(pBuf[nPos]));
		nPos	:= 47;
		n4Bytes := M_ByteSwap_REAL_TO_BYTES(M_GenerateRandom_REAL(12.0,1.0));
		M_InsertBytes_REAL(s1:=sReply, s2:=n4Bytes, nPos:=nPos);

//nPos	:= nPos + 4;
//stat.lrMotorCurrent	:= M_ByteSwapFLOAT(ADR(pBuf[nPos]));
		nPos	:= 51;
		n4Bytes := M_ByteSwap_REAL_TO_BYTES(M_GenerateRandom_REAL(12.1,0.09));
		M_InsertBytes_REAL(s1:=sReply, s2:=n4Bytes, nPos:=nPos);

//nPos	:= nPos + 4;
//stat.lrHoursOfOperation	:= M_ByteSwapFLOAT(ADR(pBuf[nPos]));
		nPos	:= 55;
		n4Bytes := M_ByteSwap_REAL_TO_BYTES(M_GenerateRandom_REAL(1633.3,0.0));
		M_InsertBytes_REAL(s1:=sReply, s2:=n4Bytes, nPos:=nPos);


//nPos	:= nPos + 4;
//stat.nPressureScale	:= M_ByteSwapINT(ADR(pBuf[nPos]));
		nPos	:= 59;
		n2Bytes := M_ByteSwap_INT_TO_BYTES(1);
		M_InsertBytes_INT(s1:=sReply, s2:=n2Bytes, nPos:=nPos);

//nPos	:= nPos + 2;
//stat.nTempScale	:= M_ByteSwapINT(ADR(pBuf[nPos]));
		nPos	:= 61;
		n2Bytes := M_ByteSwap_INT_TO_BYTES(1);
		M_InsertBytes_INT(s1:=sReply, s2:=n2Bytes, nPos:=nPos);

//nPos	:= nPos + 2;
//pPtr	:= ADR(pBuf[nPos]);
//stat.nPanelSerialNumber	:= pPtr^;
		nPos	:= 63;
		n2Bytes := M_ByteSwap_UINT_TO_BYTES(50464);
		M_InsertBytes_INT(s1:=sReply, s2:=n2Bytes, nPos:=nPos);

//nPos	:= nPos + 2;
//stat.nModelMajorMinor	:= M_ByteSwapINT(ADR(pBuf[nPos]));
		nPos	:= 65;
		n2Bytes := M_ByteSwap_INT_TO_BYTES(539);
		M_InsertBytes_INT(s1:=sReply, s2:=n2Bytes, nPos:=nPos);

	END_IF


	// TODO
	// Calculate CRC for the first 6 bytes
	//	crc	:= M_CRC(ADR(cmd),6);
	
	FOR i:=0 TO 254 DO
		sReply1[i]	:= sReply[i];
	END_FOR

	M_GetSimReply := sReply1;
END_IF
END_METHOD

END_FUNCTION_BLOCK

// ---- POUs/Sensors/FB_CRYO_PRESSURE.TcPOU
//
// This FB reads preasure using up to two PKR 250 sensors, 
// i.e. two instances of FB_CRYO_SENSOR_PKR250.
// The resulting value is a combination of values from available/valid sensors.
// Provides status of each sensor.
// For more info, see method M_SetStatus().
//
FUNCTION_BLOCK FB_CRYO_PRESSURE
VAR_INPUT
	// IMPORTANT NOTE:
	// 		It is assumed that both pressure sensors are of same type.
	//		So, all configuration parameters are same for both sensors.
	//
	{attribute 'OPC.UA.DA' := '0'}
	// Scale factors for each sensor bits -> Volt, U = raw / scale. 
	// Default for 16-bit, +-10V or 0..10V AI: 2^16/10/2 = 3276.8 bit
	in_lrBitsPerVolt_1:	LREAL := 3276.8;	// Scale factor, U = raw / scale. Default 3276.8
	{attribute 'OPC.UA.DA' := '0'}
	in_lrBitsPerVolt_2:	LREAL := 3276.8;	// Scale factor, U = raw / scale. Default 3276.8

	{attribute 'OPC.UA.DA' := '0'}
	in_nType_1:	E_CRYO_SENSOR_TYPE_PRESS	:= E_CRYO_SENSOR_TYPE_PRESS.PKR_250;
	{attribute 'OPC.UA.DA' := '0'}
	in_nType_2:	E_CRYO_SENSOR_TYPE_PRESS	:= E_CRYO_SENSOR_TYPE_PRESS.PKR_250;
	
	
	{attribute 'OPC.UA.DA' := '0'}
	in_lrLimitInVac:	LREAL := 100.0;		// Below this value, the pressure is vacuum
	{attribute 'OPC.UA.DA' := '0'}
	in_lrLimitGoodVac:	LREAL := 10.0E-4;	// Below this value, vacuum is good
	
END_VAR
VAR
	{attribute 'OPC.UA.DA' := '1'}
	Pressure1:	FB_CRYO_SENSOR_PRESSURE;
	{attribute 'OPC.UA.DA' := '1'}
	Pressure2:	FB_CRYO_SENSOR_PRESSURE;
	
	stat:		T_CRYO_PRESSURE_STATUS;	// Complete status
END_VAR

// Get status of two vacuum gauges
M_ReadSensors();

// Set the calculated vacuum pressure
M_SetStatus();

// Get status for both vacuum gauges
METHOD M_ReadSensors
VAR_INPUT
END_VAR
Pressure1(	
	in_nType			:= in_nType_1,
	in_lrBitsPerVolt	:= in_lrBitsPerVolt_1);

Pressure2(	
	in_nType			:= in_nType_2,
	in_lrBitsPerVolt	:= in_lrBitsPerVolt_2);
END_METHOD

// Calculate pressure based on the status of the two sensors
METHOD M_SetStatus
VAR_INPUT
END_VAR
VAR
	lrTmp:		LREAL;	// Temporary var
END_VAR
//
// Determine validity and calculate pressure in user units, i.e. mbar
//
IF Pressure1.stat.bValid  AND  Pressure2.stat.bValid  THEN
	// If any of the two readings are in range, the reading is in range.
	stat.bInRange	:= (Pressure1.stat.bValueInRange  OR  Pressure2.stat.bValueInRange);
	stat.bValid			:= TRUE;
	stat.bWarningSens1	:= FALSE;
	stat.bWarningSens2	:= FALSE;
	
	// Are the readings within 10% from each other
	IF Pressure2.stat.lrPressure > 0.0 THEN
		lrTmp	:= Pressure1.stat.lrPressure / Pressure2.stat.lrPressure;
	ELSE
		lrTmp	:= 0.0;	// Dummy, just to take the higher pressure.
	END_IF
	IF lrTmp > 0.9 AND lrTmp < 1.1  THEN
		// Get the average of the two
		stat.lrPressure	:= (Pressure1.stat.lrPressure + Pressure2.stat.lrPressure) / 2;
	ELSE
		// Get the higher value
		stat.lrPressure	:= MAX(Pressure1.stat.lrPressure, Pressure2.stat.lrPressure);
	END_IF
ELSIF Pressure1.stat.bValid  AND  NOT Pressure2.stat.bValid  THEN
	// Reading of one sensor is OK.
	// However, we set a warning.
	stat.bInRange		:= Pressure1.stat.bValueInRange;
	stat.bValid			:= TRUE;
	stat.bWarningSens1	:= FALSE;
	stat.bWarningSens2	:= TRUE;
	// Take the reading of the first sensor
	stat.lrPressure		:= Pressure1.stat.lrPressure;
ELSIF NOT Pressure1.stat.bValid  AND  Pressure2.stat.bValid  THEN
	// Reading of one sensor is OK.
	// However, we set a warning.
	stat.bInRange		:= Pressure2.stat.bValueInRange;
	stat.bValid			:= TRUE;
	stat.bWarningSens1	:= TRUE;
	stat.bWarningSens2	:= FALSE;
	// Take the reading of the second sensor
	stat.lrPressure		:= Pressure2.stat.lrPressure;
ELSE
	// Both readings are not valid.
	// Reading is not valid.
	stat.bInRange		:= FALSE;
	stat.bValid			:= FALSE;
	stat.bWarningSens1	:= TRUE;
	stat.bWarningSens2	:= TRUE;
	stat.lrPressure		:= 0.0;	// Dummy if reading not valid
END_IF


//
// Set vacuum state based on the pressure level
//
IF NOT stat.bValid  THEN
	stat.bInVacuum		:= FALSE;
	stat.bVacuumGood	:= FALSE;
ELSE
	// 	Check the vacuum levels
	IF stat.lrPressure < in_lrLimitGoodVac  THEN
		stat.bInVacuum		:= TRUE;
		stat.bVacuumGood	:= TRUE;
	ELSIF stat.lrPressure < in_lrLimitInVac  THEN
		stat.bInVacuum		:= TRUE;
		stat.bVacuumGood	:= FALSE;
	ELSE
		stat.bInVacuum		:= FALSE;
		stat.bVacuumGood	:= FALSE;
	END_IF
END_IF
END_METHOD

END_FUNCTION_BLOCK

// ---- POUs/Sensors/FB_CRYO_SENSOR_PRESSURE.TcPOU
FUNCTION_BLOCK FB_CRYO_SENSOR_PRESSURE EXTENDS FB_CRYO_SENSOR_BASE
VAR_INPUT
	{attribute 'OPC.UA.DA' := '0'}
	in_nType:	E_CRYO_SENSOR_TYPE_PRESS;
	{attribute 'OPC.UA.DA' := '0'}
	// Scale factor bits -> Volt, U = raw / scale. 
	// Default for 16-bit, +-10V or 0..10V AI: 2^16/10/2 = 3276.8 bit
	in_lrBitsPerVolt:	LREAL := 3276.8;	// Scale factor, U = raw / scale. Default 3276.8
	{attribute 'OPC.UA.DA' := '0'}
	in_nSampleTime:		UINT := 2000;	// Time for average read sample [ms]
END_VAR
VAR_OUTPUT
END_VAR
VAR
	{attribute 'OPC.UA.DA' := '1'}
	stat:	T_CRYO_SENSOR_STATUS_PRESS;	// Complete status

	// Timers 
	{attribute 'OPC.UA.DA' := '0'}
	fbReadTimer:	TON; (* General Timeout *)

	// Misc internal vars
	{attribute 'OPC.UA.DA' := '0'}
	nCount:			UINT := 0;		// Number of effective samples
	{attribute 'OPC.UA.DA' := '0'}
	bReadStarted:	BOOL := FALSE;	// Used for initial trigger of the read timer
	{attribute 'OPC.UA.DA' := '0'}
	lrVoltageSum:	LREAL := 0.0;	// Total sum of Valid voltages during sample time.
	{attribute 'OPC.UA.DA' := '0'}
	lrVoltageAve:	LREAL := 0.0;	// Average voltage over in_nSampleTime
END_VAR

// Set references
RefStat	REF=stat;

IF NOT bReadStarted THEN
	bReadStarted	:= TRUE;
	fbReadTimer(IN:=FALSE);
END_IF
fbReadTimer(IN:=TRUE,PT:=UINT_TO_TIME(in_nSampleTime));


// Execute the base FB
SUPER^();

// Calculate pressure based on the status in input value
METHOD M_SetStatus
VAR_INPUT
END_VAR
VAR
END_VAR
// Set pressure sensor type
stat.nType	:= in_nType;

// Update validity and the pressure in user units, i.e. mbar
CASE in_nType OF
	E_CRYO_SENSOR_TYPE_PRESS.PKR_250:
		M_SetStatus_PKR_250();
	E_CRYO_SENSOR_TYPE_PRESS.PKR_360:
		M_SetStatus_PKR_360();
	E_CRYO_SENSOR_TYPE_PRESS.CMR_361:
		M_SetStatus_CMR_361();
	E_CRYO_SENSOR_TYPE_PRESS.WRG_D_NW25:
		M_SetStatus_WRG_D_NW25();
END_CASE
END_METHOD

// Calculate pressure based on the status in input value
METHOD M_SetStatus_CMR_361
VAR_INPUT
END_VAR
VAR
	// Pfeiffer CMR361 Conversion Volt -> mbar.
	// P = (U - 1) * C1 * C2 [mbar]
	// Defaults are for Pfeiffer CMR361 (note: C1 = 0.125, C2=FullScale = 1000): 
	// P = (U - 1) * 0.125 * 1000.0 = (U-1) * 125[mbar]
	
	lrVoltage:		LREAL;	
END_VAR
// Update validity and the pressure in user units, i.e. mbar.

// Sum up all valid voltages in the range (1.0..9.8V].
IF NOT stat.bInputError  AND  stat.bInputValid  AND stat.bInputActive  THEN
	// Convert bits -> Volt
	lrVoltage	:= i_nValue / in_lrBitsPerVolt;

	// If reading is (1.0..9.8V], add the voltage to the Sum
	IF lrVoltage > 1.0  AND  lrVoltage <= 9.8 THEN
		nCount			:= nCount + 1;
		lrVoltageSum	:= lrVoltageSum + lrVoltage;
	END_IF
END_IF


// If the timer has expired, calculate the average voltage/pressure.
// Also, restart timer, and reset the counter and lrVoltageSum.
IF fbReadTimer.Q THEN
	fbReadTimer(IN:=FALSE);	// Reset timer
	IF nCount > 0 THEN
		stat.lrVoltage	:= lrVoltageSum / nCount;	// Average voltage
	ELSE
		stat.lrVoltage	:= 0.0;	// Dummy voltage - error.
	END_IF
	nCount			:= 0;
	lrVoltageSum	:= 0.0;

	// Convert Volt -> Pressure [mbar]
	// Measuring range [0.1...1100mbar] = [1.0008...9.8V]
	stat.lrPressure		:= (stat.lrVoltage - 1.0) * 125.0;

	// Check the validity of the measurement.
	// < 0.4 V - ERROR, sensor problem, Underrange
	// < 1.0V - NOT Valid, Underrange
	// < 1.0008V (0.1mbar) - Valid, underrange
	//   1.0008V (0.1mbar) .. 9.8V (1100mbar) - Valid, in range
	// > 9.8V (1100mbar) - NOT Valid, Overrange
	IF stat.lrVoltage <= 0.4	THEN
		stat.bError				:= TRUE;
		stat.bValid				:= FALSE;
		stat.bValueInRange		:= FALSE;
		stat.bValueUnderrange	:= TRUE;
		stat.bValueOverrange	:= FALSE;
	ELSIF stat.lrVoltage <= 1.0	THEN
		stat.bError				:= FALSE;
		stat.bValid				:= FALSE;
		stat.bValueInRange		:= FALSE;
		stat.bValueUnderrange	:= TRUE;
		stat.bValueOverrange	:= FALSE;
	ELSIF stat.lrVoltage < 1.0008	THEN
		stat.bError				:= FALSE;
		stat.bValid				:= TRUE;
		stat.bValueInRange		:= FALSE;
		stat.bValueUnderrange	:= TRUE;
		stat.bValueOverrange	:= FALSE;
	ELSIF stat.lrVoltage <= 9.8	THEN
		stat.bError				:= FALSE;
		stat.bValid				:= TRUE;
		stat.bValueInRange		:= TRUE;
		stat.bValueUnderrange	:= FALSE;
		stat.bValueOverrange	:= FALSE;
	ELSE
		stat.bError				:= TRUE;
		stat.bValid				:= FALSE;
		stat.bValueInRange		:= FALSE;
		stat.bValueUnderrange	:= FALSE;
		stat.bValueOverrange	:= TRUE;
	END_IF

END_IF
END_METHOD

// Calculate pressure based on the status in input value
METHOD M_SetStatus_PKR_250
VAR_INPUT
END_VAR
VAR
	// Pfeiffer PKR250/251 Conversion Volt -> mbar.
	// P = 10^(C1 * U - C2).
	// Defaults are for Pfeiffer PKR250/251 (note: C1 = 1.667, C2 = d = 11.33): 
	// P = 10^(1.667 * U - 11.33)
	// Valid range for U is 1.8-8.6
	//
	
	lrVoltage:		LREAL;
END_VAR
// Update validity and the pressure in user units, i.e. mbar.

// Sum up all valid voltages in the range [1.4..9.5V].
IF NOT stat.bInputError  AND  stat.bInputValid  AND stat.bInputActive  THEN
	// Convert bits -> Volt
	lrVoltage	:= i_nValue / in_lrBitsPerVolt;

	// If reading is [1.4..9.5V], add the voltage to the Sum
	IF lrVoltage >= 1.4  AND  lrVoltage <= 9.5 THEN
		nCount			:= nCount + 1;
		lrVoltageSum	:= lrVoltageSum + lrVoltage;
	END_IF
END_IF


// If the timer has expired, calculate the average voltage/pressure.
// Also, restart timer, and reset the counter and lrVoltageSum.
IF fbReadTimer.Q THEN
	fbReadTimer(IN:=FALSE);	// Reset timer
	IF nCount > 0 THEN
		stat.lrVoltage	:= lrVoltageSum / nCount;	// Average voltage
	ELSE
		stat.lrVoltage	:= 0.0;	// Dummy voltage - error.
	END_IF
	nCount			:= 0;
	lrVoltageSum	:= 0.0;

	// Convert Volt -> Pressure [mbar]
	// Measuring range [0.1...1100mbar] = [1.0008...9.8V]
	stat.lrPressure		:= EXPT(10.0, (1.667 * stat.lrVoltage - 11.33));

	// Check the validity of the measurement.
	// < 0.5 V - ERROR, sensor problem, Underrange
	// < 1.4V (1E-09mbar)- NOT Valid, Underrange
	// < 1.76V (4E-09mbar) - Valid, underrange
	//   1.76V (4E-09mbar) .. 8.6V (1014mbar) - Valid, in range
	// < 9.5V (1014mbar) - Valid, Overrange, fixed pressure to 1014mbar
	// >= 9.5V  - NOT Valid, Overrange
	IF stat.lrVoltage <= 0.5	THEN
		stat.bError				:= TRUE;
		stat.bValid				:= FALSE;
		stat.bValueInRange		:= FALSE;
		stat.bValueUnderrange	:= TRUE;
		stat.bValueOverrange	:= FALSE;
	ELSIF stat.lrVoltage < 1.4	THEN
		stat.bError				:= FALSE;
		stat.bValid				:= FALSE;
		stat.bValueInRange		:= FALSE;
		stat.bValueUnderrange	:= TRUE;
		stat.bValueOverrange	:= FALSE;
	ELSIF stat.lrVoltage < 1.76	THEN
		stat.bError				:= FALSE;
		stat.bValid				:= TRUE;
		stat.bValueInRange		:= FALSE;
		stat.bValueUnderrange	:= TRUE;
		stat.bValueOverrange	:= FALSE;
	ELSIF stat.lrVoltage <= 8.6	THEN
		stat.bError				:= FALSE;
		stat.bValid				:= TRUE;
		stat.bValueInRange		:= TRUE;
		stat.bValueUnderrange	:= FALSE;
		stat.bValueOverrange	:= FALSE;
	ELSIF stat.lrVoltage <= 9.5	THEN
		stat.bError				:= FALSE;
		stat.bValid				:= TRUE;
		stat.bValueInRange		:= FALSE;
		stat.bValueUnderrange	:= FALSE;
		stat.bValueOverrange	:= TRUE;
		stat.lrPressure			:= 1014.0;
	ELSE
		stat.bError				:= TRUE;
		stat.bValid				:= FALSE;
		stat.bValueInRange		:= FALSE;
		stat.bValueUnderrange	:= FALSE;
		stat.bValueOverrange	:= TRUE;
	END_IF

END_IF
END_METHOD

// Calculate pressure based on the status in input value
METHOD M_SetStatus_PKR_360
VAR_INPUT
END_VAR
VAR
	// Pfeiffer PKR360 Conversion Volt -> mbar.
	// P = 10^(C1 * U - C2).
	// Defaults are for Pfeiffer PKR250/251 (note: C1 = 1.667, C2 = d = 11.33): 
	// P = 10^(1.667 * U - 11.33)
	// Valid range for U is 1.397-8.6 (up to 9.5 fixed to 1014 mbar in SW)
	//
	
	lrVoltage:		LREAL;
END_VAR
// Update validity and the pressure in user units, i.e. mbar.

// Sum up all valid voltages in the range [1.397 .. 9.5V].
IF NOT stat.bInputError  AND  stat.bInputValid  AND stat.bInputActive  THEN
	// Convert bits -> Volt
	lrVoltage	:= i_nValue / in_lrBitsPerVolt;

	// If reading is [1.4..9.5V], add the voltage to the Sum
	IF lrVoltage >= 1.397  AND  lrVoltage <= 9.5 THEN
		nCount			:= nCount + 1;
		lrVoltageSum	:= lrVoltageSum + lrVoltage;
	END_IF
END_IF


// If the timer has expired, calculate the average voltage/pressure.
// Also, restart timer, and reset the counter and lrVoltageSum.
IF fbReadTimer.Q THEN
	fbReadTimer(IN:=FALSE);	// Reset timer
	IF nCount > 0 THEN
		stat.lrVoltage	:= lrVoltageSum / nCount;	// Average voltage
	ELSE
		stat.lrVoltage	:= 0.0;	// Dummy voltage - error.
	END_IF
	nCount			:= 0;
	lrVoltageSum	:= 0.0;

	// Convert Volt -> Pressure [mbar]
	// Measuring range [0.1...1100mbar] = [1.0008...9.5V]
	stat.lrPressure		:= EXPT(10.0, (1.667 * stat.lrVoltage - 11.33));

	// Check the validity of the measurement.
	// < 1.217 V - ERROR, sensor problem, Underrange
	// < 1.397V (1E-09mbar)- NOT Valid, Underrange
	//   8.6V (4E-09mbar) .. 8.6V (1014mbar) - Valid, in range
	// < 9.5V (1014mbar) - Valid, Overrange, fixed pressure to 1014mbar
	// >= 9.5V  - NOT Valid, Overrange
	IF stat.lrVoltage <= 1.217	THEN
		stat.bError				:= TRUE;
		stat.bValid				:= FALSE;
		stat.bValueInRange		:= FALSE;
		stat.bValueUnderrange	:= TRUE;
		stat.bValueOverrange	:= FALSE;
	ELSIF stat.lrVoltage < 1.397	THEN
		stat.bError				:= FALSE;
		stat.bValid				:= FALSE;
		stat.bValueInRange		:= FALSE;
		stat.bValueUnderrange	:= TRUE;
		stat.bValueOverrange	:= FALSE;
	ELSIF stat.lrVoltage <= 8.6	THEN
		stat.bError				:= FALSE;
		stat.bValid				:= TRUE;
		stat.bValueInRange		:= TRUE;
		stat.bValueUnderrange	:= FALSE;
		stat.bValueOverrange	:= FALSE;
	ELSIF stat.lrVoltage <= 9.5	THEN
		stat.bError				:= FALSE;
		stat.bValid				:= TRUE;
		stat.bValueInRange		:= FALSE;
		stat.bValueUnderrange	:= FALSE;
		stat.bValueOverrange	:= TRUE;
		stat.lrPressure			:= 1014.0;
	ELSE
		stat.bError				:= TRUE;
		stat.bValid				:= FALSE;
		stat.bValueInRange		:= FALSE;
		stat.bValueUnderrange	:= FALSE;
		stat.bValueOverrange	:= TRUE;
	END_IF

END_IF
END_METHOD

// Calculate pressure based on the status in input value
METHOD M_SetStatus_WRG_D_NW25
VAR_INPUT
END_VAR
VAR
	// Edwards WRG-D-NW25 Conversion Volt -> mbar.
	// Range 10^-9 .. 100
	// P = 10^(C1 * U - C2).
	// P = 10^(1.5 * U - 12.0)
	// Valid range for U is 2.0-10.0
	//
	
	lrVoltage:		LREAL;
END_VAR
// Update validity and the pressure in user units, i.e. mbar.

// Sum up all valid voltages in the range [2.0..10.0V].
IF NOT stat.bInputError  AND  stat.bInputValid  AND stat.bInputActive  THEN
	// Convert bits -> Volt
	lrVoltage	:= i_nValue / in_lrBitsPerVolt;

	// If reading is [2.0..10.0V], add the voltage to the Sum
	IF lrVoltage >= 2.0  AND  lrVoltage <= 10.0 THEN
		nCount			:= nCount + 1;
		lrVoltageSum	:= lrVoltageSum + lrVoltage;
	END_IF
END_IF


// If the timer has expired, calculate the average voltage/pressure.
// Also, restart timer, and reset the counter and lrVoltageSum.
IF fbReadTimer.Q THEN
	fbReadTimer(IN:=FALSE);	// Reset timer
	IF nCount > 0 THEN
		stat.lrVoltage	:= lrVoltageSum / nCount;	// Average voltage
	ELSE
		stat.lrVoltage	:= 0.0;	// Dummy voltage - error.
	END_IF
	nCount			:= 0;
	lrVoltageSum	:= 0.0;

	// Convert Volt -> Pressure [mbar]
	// Measuring range [0.1...1000mbar] = [2.0...10.0V]
	stat.lrPressure		:= EXPT(10.0, (1.5 * stat.lrVoltage - 12.0));

	// Check the validity of the measurement.
	// < 1.5 V - ERROR, sensor problem, Underrange
	// < 2.0V (1E-09mbar)- NOT Valid, Underrange
	// < 10.0V (1000mbar) - Valid
	// < 10.15V (1678mbar) - NOT Valid, Overrange
	// >= 10.15V  - Error, Overrange
	IF stat.lrVoltage < 1.5	THEN
		stat.bError				:= TRUE;
		stat.bValid				:= FALSE;
		stat.bValueInRange		:= FALSE;
		stat.bValueUnderrange	:= TRUE;
		stat.bValueOverrange	:= FALSE;
	ELSIF stat.lrVoltage < 2.0	THEN
		stat.bError				:= FALSE;
		stat.bValid				:= FALSE;
		stat.bValueInRange		:= FALSE;
		stat.bValueUnderrange	:= TRUE;
		stat.bValueOverrange	:= FALSE;
	ELSIF stat.lrVoltage <= 10.0	THEN
		stat.bError				:= FALSE;
		stat.bValid				:= TRUE;
		stat.bValueInRange		:= TRUE;
		stat.bValueUnderrange	:= FALSE;
		stat.bValueOverrange	:= FALSE;
	ELSIF stat.lrVoltage <= 10.15	THEN
		stat.bError				:= FALSE;
		stat.bValid				:= FALSE;
		stat.bValueInRange		:= FALSE;
		stat.bValueUnderrange	:= FALSE;
		stat.bValueOverrange	:= TRUE;
	ELSE
		stat.bError				:= TRUE;
		stat.bValid				:= FALSE;
		stat.bValueInRange		:= FALSE;
		stat.bValueUnderrange	:= FALSE;
		stat.bValueOverrange	:= TRUE;
	END_IF

END_IF
END_METHOD

END_FUNCTION_BLOCK

// ---- POUs/Sensors/FB_CRYO_SENSOR_BASE.TcPOU
FUNCTION_BLOCK FB_CRYO_SENSOR_BASE
VAR_INPUT
END_VAR
VAR
	{attribute 'OPC.UA.DA' := '0'}
	i_nStatus	AT %I*: UINT;
	{attribute 'OPC.UA.DA' := '0'}
	i_nValue	AT%I*:	INT;
	
	{attribute 'OPC.UA.DA' := '0'}
	bStarted:		BOOL := FALSE;
	{attribute 'OPC.UA.DA' := '0'}
	toggleTimer:	TON;		// Timer for PDO (alive) toggle
	{attribute 'OPC.UA.DA' := '0'}
	toggleTrig:		R_TRIG;		// PDO (alive) toggle detection
	
	RefStat: 	REFERENCE TO T_CRYO_SENSOR_STATUS;
END_VAR

// Get the raw reading and the status of the input channel
M_ReadSensor();

// Calculate value and validity
M_SetStatus();

// Get input channel status and the raw reading
METHOD M_ReadSensor
VAR_INPUT
END_VAR
// Get input channel status
RefStat.bInputUnder	:= (i_nStatus AND 2#0000_0000_0000_0001) <> 0;
RefStat.bInputOver	:= (i_nStatus AND 2#0000_0000_0000_0010) <> 0;
RefStat.bInputError	:= (i_nStatus AND 2#0000_0000_0100_0000) <> 0;
RefStat.bInputToggle:= (i_nStatus AND 2#1000_0000_0000_0000) <> 0;
RefStat.bInputValid	:= (i_nStatus AND 2#0100_0000_0000_0000)  = 0;	// 0 -> PDO OK

// Get the raw reading
RefStat.nRawValue	:= i_nValue;

//
// Check if the terminal is alive.
// Start the time that will expire in 3 sec.
// If bToggle bit triggers before the timer expires, 
// this is the sign that the terminal is alive.
//
IF NOT bStarted THEN
	bStarted	:= TRUE;
	toggleTimer(IN:=FALSE);
END_IF
toggleTimer(IN:=TRUE,PT:=T#3S);
toggleTrig(CLK:=RefStat.bInputToggle);

IF toggleTrig.Q THEN
	// bToggle bit has triggered. Terminal is alive.
	RefStat.bInputActive	:= TRUE;
	// Restart the timer
	toggleTimer(IN:=FALSE);
ELSIF toggleTimer.Q THEN
	// bInputToggle bit has not triggered within 3 sec. Terminal is NOT alive.
	RefStat.bInputActive	:= FALSE;
	// Restart the timer
	toggleTimer(IN:=FALSE);
END_IF
END_METHOD

METHOD M_SetStatus
VAR_INPUT
END_VAR
// TODO USER: Implement the method.
END_METHOD

END_FUNCTION_BLOCK

// ---- POUs/Sensors/FB_CRYO_TEMPERATURE.TcPOU
//
// This FB reads temperature using up to two sensors, i.e. instances of FB_CRYO_PT100.
// The resulting value is the temperature of the first available/valid sensor.
// Provides status of each sensor.
//
FUNCTION_BLOCK FB_CRYO_TEMPERATURE
VAR_INPUT
	{attribute 'OPC.UA.DA' := '0'}
	in_bSimulation:	BOOL	:= FALSE;	// If TRUE, the temperature value is simulated.
	
	{attribute 'OPC.UA.DA' := '0'}
	in_nType_1:				E_CRYO_SENSOR_TYPE_TEMP	:= E_CRYO_SENSOR_TYPE_TEMP.PT100;
	{attribute 'OPC.UA.DA' := '0'}
	in_nType_2:				E_CRYO_SENSOR_TYPE_TEMP	:= E_CRYO_SENSOR_TYPE_TEMP.PT100;
	{attribute 'OPC.UA.DA' := '0'}
	in_lrScale_1:			LREAL := 0.1;	// Scale factor, T = raw * scale. Default 0.1
	{attribute 'OPC.UA.DA' := '0'}
	in_lrScale_2:			LREAL := 0.1;	// Scale factor, T = raw * scale. Default 0.1
	{attribute 'OPC.UA.DA' := '0'}
	in_bIgnoreUnderrange_1:	BOOL := TRUE;	// If True, underrange is also valid
	{attribute 'OPC.UA.DA' := '0'}
	in_bIgnoreUnderrange_2:	BOOL := TRUE;	// If True, underrange is also valid
	{attribute 'OPC.UA.DA' := '0'}
	in_nRampPeriodSec:		UDINT := 60;	// Ramp measurement period [sec]. Default 60 sec.
	
END_VAR
VAR
	{attribute 'OPC.UA.DA' := '1'}
	Temperature1:	FB_CRYO_SENSOR_TEMPERATURE;
	{attribute 'OPC.UA.DA' := '1'}
	Temperature2:	FB_CRYO_SENSOR_TEMPERATURE;
	
	{attribute 'OPC.UA.DA' := '1'}
	stat:			T_CRYO_TEMPERATURE_STATUS;
END_VAR

// Get the raw reading and the status of the input channel
M_ReadSensors();

// Calculate temperatures and validity
M_SetStatus();

METHOD M_GetTemperatureFromLakeshore
VAR_INPUT
	bValid:		BOOL;	// Flag if reading is valid
	lrTempK:	LREAL;	// Lakeshore reading in degK 
	lrTempC:	LREAL;	// Lakeshore reading in degC 
END_VAR
//
// Check if the temperature is coming from the simulator 
// of the Lakeshore temperature.
//
// The simulator reading is always valid.
// If the temperature is not linked to a simulator,
// it will not be Valid since it is not mapped at all!!!
// If simulated, Temperature1 has to be linked to the simulator.
// Temperature2 should not be used/mapped in that case.
//
IF	Temperature1.stat.bValid THEN
	// Temperature is coming from a simulator.
	stat.bValid 		:= TRUE;
	stat.bWarningSens1	:= FALSE;
	stat.bWarningSens2	:= FALSE;
	stat.lrTempK		:= Temperature1.stat.lrTempK;
	stat.lrTempC		:= Temperature1.stat.lrTempC;
ELSIF bValid THEN
	// Temperature is coming from Lakeshore and is Valid.
	stat.bValid 		:= TRUE;
	stat.bWarningSens1	:= FALSE;
	stat.bWarningSens2	:= FALSE;
	stat.lrTempK		:= lrTempK;
	stat.lrTempC		:= lrTempC;
ELSE
	// Temperature is coming from Lakeshore and is NOT Valid.
	stat.bValid 		:= FALSE;
	stat.bWarningSens1	:= TRUE;
	stat.bWarningSens2	:= TRUE;
	stat.lrTempK		:= 850.0;
	stat.lrTempC		:= 850.0;
END_IF
END_METHOD

// Get input channel status and the raw reading
METHOD M_ReadSensors
VAR_INPUT
END_VAR
Temperature1(	in_nType				:= in_nType_1,
				in_lrScale 				:= in_lrScale_1, 
				in_bIgnoreUnderrange	:= in_bIgnoreUnderrange_1,
				in_nRampPeriodSec		:= in_nRampPeriodSec);

Temperature2(	in_nType				:= in_nType_2,
				in_lrScale 				:= in_lrScale_2, 
				in_bIgnoreUnderrange	:= in_bIgnoreUnderrange_2,
				in_nRampPeriodSec		:= in_nRampPeriodSec);
END_METHOD

METHOD M_SetStatus
VAR_INPUT
END_VAR
VAR
	lrTmp:		LREAL;	// Temporary var
END_VAR
//
// If simulated, set the simulated value and return.
// Note: Simulated temperature is in [K] !!!
//
IF in_bSimulation THEN
	stat.bSimulated	:= TRUE;
	stat.bValid		:= TRUE;
	stat.lrTempK	:= stat.lrSimTempK;
	stat.lrTempC	:= stat.lrSimTempK - 273.15;
	RETURN;
ELSE
	stat.bSimulated	:= FALSE;
END_IF


//
// Determine validity and calculate temperature in degC and degK
//
IF Temperature1.stat.bValid  AND  Temperature2.stat.bValid  THEN
	// Reading is OK.
	stat.bValid			:= TRUE;
	stat.bWarningSens1	:= FALSE;
	stat.bWarningSens2	:= FALSE;

	// Take the reading of the first sensor if it is not underrange
	// or both readings are underrange.
	IF	NOT Temperature1.stat.bInputUnder	OR
		(Temperature1.stat.bInputUnder  AND  Temperature2.stat.bInputUnder) THEN
		// T1 - NOT underrange  OR  both underrange
		// Take T1
		stat.lrRamp		:= Temperature1.stat.lrRamp;
		stat.lrTempC	:= Temperature1.stat.lrTempC;
		stat.lrTempK	:= Temperature1.stat.lrTempK;
		stat.bInRange	:= NOT Temperature1.stat.bInputUnder;
	ELSE
		// T1 - underrange
		// T2 - NOT underrange
		// Take T2
		stat.lrRamp		:= Temperature2.stat.lrRamp;
		stat.lrTempC	:= Temperature2.stat.lrTempC;
		stat.lrTempK	:= Temperature2.stat.lrTempK;
		stat.bInRange	:= NOT Temperature2.stat.bInputUnder;
	END_IF
	
ELSIF Temperature1.stat.bValid  AND  NOT Temperature2.stat.bValid  THEN
	// Reading of sensor #1 is OK.
	// However, we set a warning for sensor #2.
	stat.bValid			:= TRUE;
	stat.bWarningSens1	:= FALSE;
	stat.bWarningSens2	:= TRUE;
	// Take the reading of the first sensor
	stat.lrRamp			:= Temperature1.stat.lrRamp;
	stat.lrTempC		:= Temperature1.stat.lrTempC;
	stat.lrTempK		:= Temperature1.stat.lrTempK;
	stat.bInRange		:= NOT Temperature1.stat.bInputUnder;
	
ELSIF NOT Temperature1.stat.bValid  AND  Temperature2.stat.bValid  THEN
	// Reading of sensor #1 is NOT OK.
	// Reading of sensor #2 is OK.
	// However, we set a warning.
	stat.bValid			:= TRUE;
	stat.bWarningSens1	:= TRUE;
	stat.bWarningSens2	:= FALSE;
	// Take the reading of the second sensor
	stat.lrRamp			:= Temperature2.stat.lrRamp;
	stat.lrTempC		:= Temperature2.stat.lrTempC;
	stat.lrTempK		:= Temperature2.stat.lrTempK;
	stat.bInRange		:= NOT Temperature2.stat.bInputUnder;
	
ELSE
	// Both readings are not valid.
	// Reading is not valid.
	stat.bInRange		:= FALSE;
	stat.bValid			:= FALSE;
	stat.bWarningSens1	:= TRUE;
	stat.bWarningSens2	:= TRUE;
	// Readings are not valid.
	// The value is not important.
	// Take the value of the first sensor.
	// It might show under/over range.
	stat.lrRamp			:= 0.0;
	stat.lrTempC		:= Temperature1.stat.lrTempC;
	stat.lrTempK		:= Temperature1.stat.lrTempK;

END_IF


//
// If the reading is valid, set the simulated value to it.
// This way, switching from normal to simulation will result in
// no jump in the value.
//
IF stat.bValid  THEN
	stat.lrSimTempK	:= stat.lrTempK;
END_IF
END_METHOD

END_FUNCTION_BLOCK

// ---- POUs/Sensors/FB_CRYO_SENSOR_TEMPERATURE.TcPOU
FUNCTION_BLOCK FB_CRYO_SENSOR_TEMPERATURE EXTENDS FB_CRYO_SENSOR_BASE
VAR_INPUT
	{attribute 'OPC.UA.DA' := '0'}
	in_nType:				E_CRYO_SENSOR_TYPE_TEMP	:= E_CRYO_SENSOR_TYPE_TEMP.PT100;
	{attribute 'OPC.UA.DA' := '0'}
	in_lrScale:				LREAL := 0.1;		// Scale factor, T = raw * scale. Default 0.1
	{attribute 'OPC.UA.DA' := '0'}
	in_bIgnoreUnderrange:	BOOL  := FALSE;		// If T, underrange will be treated as bValid.
	{attribute 'OPC.UA.DA' := '0'}
	in_nRampPeriodSec:		UDINT := 60;		// Ramp measurement period [sec]. Default 60 sec.
	// If true, temperature calculated from measured resistance.
	// With this flag active, temperature range is extended to -240 degC.
	{attribute 'OPC.UA.DA' := '0'}
	in_bResistor_1_64:		BOOL := FALSE;		
END_VAR
VAR_OUTPUT
END_VAR
VAR
	{attribute 'OPC.UA.DA' := '1'}
	stat:	T_CRYO_SENSOR_STATUS_TEMP;	// Complete status

	{attribute 'OPC.UA.DA' := '0'}
	bRampTimerStarted:	BOOL := FALSE;
	{attribute 'OPC.UA.DA' := '0'}
	rampTimer:	TON;		// Timer for calculating ramp
	
	// Lookup table when converting resistance to Celsius, range [-240..200].
	// NOTE: RTD Element in CoE of the RTD terminal, e.g., EL3201
	//       must be configured for "Resistor 1/64 Ohm..."
	//       Also, in_bResistor_1_64 must be set to TRUE.
	LookupTable:	ARRAY [0..88] OF T_CRYO_PT100_OHM2C_REC := [
			(celsius := 	-240.0	, ohm := 	0.911	),
			(celsius := 	-235.0	, ohm := 	3.150	),
			(celsius := 	-230.0	, ohm := 	5.377	),
			(celsius := 	-225.0	, ohm := 	7.594	),
			(celsius := 	-220.0	, ohm := 	9.799	),
			(celsius := 	-215.0	, ohm := 	11.995	),
			(celsius := 	-210.0	, ohm := 	14.180	),
			(celsius := 	-205.0	, ohm := 	16.356	),
			(celsius := 	-200.0	, ohm := 	18.522	),
			(celsius := 	-195.0	, ohm := 	20.679	),
			(celsius := 	-190.0	, ohm := 	22.827	),
			(celsius := 	-185.0	, ohm := 	24.967	),
			(celsius := 	-180.0	, ohm := 	27.098	),
			(celsius := 	-175.0	, ohm := 	29.221	),
			(celsius := 	-170.0	, ohm := 	31.336	),
			(celsius := 	-165.0	, ohm := 	33.444	),
			(celsius := 	-160.0	, ohm := 	35.545	),
			(celsius := 	-155.0	, ohm := 	37.638	),
			(celsius := 	-150.0	, ohm := 	39.724	),
			(celsius := 	-145.0	, ohm := 	41.804	),
			(celsius := 	-140.0	, ohm := 	43.877	),
			(celsius := 	-135.0	, ohm := 	45.945	),
			(celsius := 	-130.0	, ohm := 	48.006	),
			(celsius := 	-125.0	, ohm := 	50.061	),
			(celsius := 	-120.0	, ohm := 	52.110	),
			(celsius := 	-115.0	, ohm := 	54.155	),
			(celsius := 	-110.0	, ohm := 	56.194	),
			(celsius := 	-105.0	, ohm := 	58.227	),
			(celsius := 	-100.0	, ohm := 	60.256	),
			(celsius := 	-95.0	, ohm := 	62.280	),
			(celsius := 	-90.0	, ohm := 	64.300	),
			(celsius := 	-85.0	, ohm := 	66.315	),
			(celsius := 	-80.0	, ohm := 	68.326	),
			(celsius := 	-75.0	, ohm := 	70.332	),
			(celsius := 	-70.0	, ohm := 	72.335	),
			(celsius := 	-65.0	, ohm := 	74.333	),
			(celsius := 	-60.0	, ohm := 	76.328	),
			(celsius := 	-55.0	, ohm := 	78.319	),
			(celsius := 	-50.0	, ohm := 	80.306	),
			(celsius := 	-45.0	, ohm := 	82.290	),
			(celsius := 	-40.0	, ohm := 	84.271	),
			(celsius := 	-35.0	, ohm := 	86.248	),
			(celsius := 	-30.0	, ohm := 	88.222	),
			(celsius := 	-25.0	, ohm := 	90.192	),
			(celsius := 	-20.0	, ohm := 	92.160	),
			(celsius := 	-15.0	, ohm := 	94.124	),
			(celsius := 	-10.0	, ohm := 	96.086	),
			(celsius := 	-5.0	, ohm := 	98.044	),
			(celsius := 	0.0		, ohm := 	100.000	),
			(celsius := 	5.0		, ohm := 	101.953	),
			(celsius := 	10.0	, ohm := 	103.903	),
			(celsius := 	15.0	, ohm := 	105.850	),
			(celsius := 	20.0	, ohm := 	107.794	),
			(celsius := 	25.0	, ohm := 	109.735	),
			(celsius := 	30.0	, ohm := 	111.674	),
			(celsius := 	35.0	, ohm := 	113.610	),
			(celsius := 	40.0	, ohm := 	115.542	),
			(celsius := 	45.0	, ohm := 	117.473	),
			(celsius := 	50.0	, ohm := 	119.400	),
			(celsius := 	55.0	, ohm := 	121.324	),
			(celsius := 	60.0	, ohm := 	123.246	),
			(celsius := 	65.0	, ohm := 	125.164	),
			(celsius := 	70.0	, ohm := 	127.080	),
			(celsius := 	75.0	, ohm := 	128.992	),
			(celsius := 	80.0	, ohm := 	130.901	),
			(celsius := 	85.0	, ohm := 	132.808	),
			(celsius := 	90.0	, ohm := 	134.710	),
			(celsius := 	95.0	, ohm := 	136.610	),
			(celsius := 	100.0	, ohm := 	138.506	),
			(celsius := 	105.0	, ohm := 	140.399	),
			(celsius := 	110.0	, ohm := 	142.288	),
			(celsius := 	115.0	, ohm := 	144.173	),
			(celsius := 	120.0	, ohm := 	146.054	),
			(celsius := 	125.0	, ohm := 	147.932	),
			(celsius := 	130.0	, ohm := 	149.805	),
			(celsius := 	135.0	, ohm := 	151.674	),
			(celsius := 	140.0	, ohm := 	153.539	),
			(celsius := 	145.0	, ohm := 	155.400	),
			(celsius := 	150.0	, ohm := 	157.256	),
			(celsius := 	155.0	, ohm := 	159.107	),
			(celsius := 	160.0	, ohm := 	160.953	),
			(celsius := 	165.0	, ohm := 	162.794	),
			(celsius := 	170.0	, ohm := 	164.630	),
			(celsius := 	175.0	, ohm := 	166.460	),
			(celsius := 	180.0	, ohm := 	168.285	),
			(celsius := 	185.0	, ohm := 	170.104	),
			(celsius := 	190.0	, ohm := 	171.917	),
			(celsius := 	195.0	, ohm := 	173.723	),
			(celsius := 	200.0	, ohm := 	175.523	)];

			lrTemStep:	LREAL	:= 5.0; 	// Temperature step in the table.
			nLastIndex:	INT		:= 0;

END_VAR

// Set references
RefStat	REF=stat;

// Execute the base FB
SUPER^();

// Calculate Temperature change ramp
M_GetRamp();

METHOD M_GetRamp
VAR_INPUT
END_VAR
VAR_INST
	{attribute 'OPC.UA.DA' := '0'}
	lrRampStartTempK:	LREAL;	// Temperature at start of ramp timer [K]
END_VAR
VAR
	nRampPeriodSec:		UDINT;	// Ramp measurement period [sec].
END_VAR
IF NOT bRampTimerStarted THEN
	bRampTimerStarted	:= TRUE;
	lrRampStartTempK	:= stat.lrTempK;
	rampTimer(IN:=FALSE);
END_IF

// Execute timer.
// Ramp measurement period should be > 0
nRampPeriodSec	:= in_nRampPeriodSec;
IF nRampPeriodSec = 0 THEN
	nRampPeriodSec	:= 60;
END_IF
rampTimer(IN:=TRUE,PT:=UDINT_TO_TIME(nRampPeriodSec)*1000);

// Calculate ramp at time expiry
IF rampTimer.Q THEN
	// Calculate the temperature ramp per minute
	IF stat.bValid THEN
		stat.lrRamp	:= (stat.lrTempK - lrRampStartTempK) * 60.0 / nRampPeriodSec;
	ELSE
		stat.lrRamp	:= 0.0;
	END_IF

	// Current temperature is the starting value of the ramp
	lrRampStartTempK	:= stat.lrTempK;

	// Restart the timer
	rampTimer(IN:=FALSE);
END_IF
END_METHOD

